LIN {X 0,Y 316.266,Z 772.149,A -85,B 0,C 180,E1 7195.232,E2 7195.232} C_VEL
LIN {X 0,Y 308.855,Z 793.821,A -85,B 0,C 180,E1 7194.701,E2 7194.701} C_VEL
LIN {X 0,Y 300.069,Z 815.244,A -85,B 0,C 180,E1 7194.002,E2 7194.002} C_VEL
LIN {X 0,Y 290.008,Z 835.58,A -85,B 0,C 180,E1 7193.134,E2 7193.134} C_VEL
LIN {X 0,Y 278.14,Z 856.299,A -85,B 0,C 180,E1 7191.998,E2 7191.998} C_VEL
LIN {X 0,Y 266.399,Z 874.047,A -85,B 0,C 180,E1 7190.75,E2 7190.75} C_VEL
LIN {X 0,Y 252.026,Z 893.205,A -85,B 0,C 180,E1 7189.023,E2 7189.023} C_VEL
LIN {X 0,Y 238.567,Z 909.092,A -85,B 0,C 180,E1 7187.167,E2 7187.167} C_VEL
LIN {X 0,Y 222.897,Z 925.612,A -85,B 0,C 180,E1 7184.652,E2 7184.652} C_VEL
LIN {X 0,Y 207.871,Z 939.883,A -85,B 0,C 180,E1 7181.782,E2 7181.782} C_VEL
LIN {X 0,Y 191.846,Z 953.573,A -85,B 0,C 180,E1 7178.064,E2 7178.064} C_VEL
LIN {X 0,Y 176.404,Z 965.739,A -85,B 0,C 180,E1 7173.567,E2 7173.567} C_VEL
LIN {X 0,Y 161.53,Z 976.411,A -85,B 0,C 180,E1 7167.988,E2 7167.988} C_VEL
LIN {X 0,Y 147.743,Z 985.877,A -85,B 0,C 180,E1 7160.997,E2 7160.997} C_VEL
LIN {X 0,Y 136.959,Z 993.036,A -85,B 0,C 180,E1 7153.329,E2 7153.329} C_VEL
LIN {X 0,Y 127.495,Z 999.606,A -85,B 0,C 180,E1 7142.954,E2 7142.954} C_VEL
LIN {X 0,Y 122.646,Z 1003.525,A -85,B 0,C 180,E1 7133.543,E2 7133.543} C_VEL
LIN {X 0,Y 120.303,Z 1006.266,A -85,B 0,C 180,E1 7122.968,E2 7122.968} C_VEL
LIN {X 0,Y 120.046,Z 1007.285,A -85,B 0,C 180,E1 7114.778,E2 7114.778} C_VEL
LIN {X 0,Y 120.078,Z 1007.432,A -85,B 0,C 180,E1 7108.093,E2 7108.093} C_VEL
LIN {X 0,Y 120.087,Z 1006.85,A -85,B 0,C 180,E1 7100.9,E2 7100.9} C_VEL
LIN {X 0,Y 121.024,Z 1005.17,A -85,B 0,C 180,E1 7092.204,E2 7092.204} C_VEL
LIN {X 0,Y 124.46,Z 1001.976,A -85,B 0,C 180,E1 7082.233,E2 7082.233} C_VEL
LIN {X 0,Y 131.486,Z 996.711,A -85,B 0,C 180,E1 7071.986,E2 7071.986} C_VEL
LIN {X 0,Y 141.32,Z 990.14,A -85,B 0,C 180,E1 7063.228,E2 7063.228} C_VEL
LIN {X 0,Y 153.783,Z 981.683,A -85,B 0,C 180,E1 7055.648,E2 7055.648} C_VEL
LIN {X 0,Y 168.407,Z 971.472,A -85,B 0,C 180,E1 7049.233,E2 7049.233} C_VEL
LIN {X 0,Y 183.206,Z 960.371,A -85,B 0,C 180,E1 7044.315,E2 7044.315} C_VEL
LIN {X 0,Y 199.948,Z 946.664,A -85,B 0,C 180,E1 7039.95,E2 7039.95} C_VEL
LIN {X 0,Y 215.947,Z 932.296,A -85,B 0,C 180,E1 7036.603,E2 7036.603} C_VEL
LIN {X 0,Y 231.694,Z 916.357,A -85,B 0,C 180,E1 7033.869,E2 7033.869} C_VEL
LIN {X 0,Y 247.003,Z 899.128,A -85,B 0,C 180,E1 7031.627,E2 7031.627} C_VEL
LIN {X 0,Y 260.107,Z 882.465,A -85,B 0,C 180,E1 7029.961,E2 7029.961} C_VEL
LIN {X 0,Y 274.246,Z 862.079,A -85,B 0,C 180,E1 7028.385,E2 7028.385} C_VEL
LIN {X 0,Y 285.918,Z 842.77,A -85,B 0,C 180,E1 7027.232,E2 7027.232} C_VEL
LIN {X 0,Y 296.695,Z 821.891,A -85,B 0,C 180,E1 7026.268,E2 7026.268} C_VEL
LIN {X 0,Y 305.842,Z 801.227,A -85,B 0,C 180,E1 7025.53,E2 7025.53} C_VEL
LIN {X 0,Y 313.42,Z 780.232,A -85,B 0,C 180,E1 7024.959,E2 7024.959} C_VEL
LIN {X 0,Y 320.064,Z 757.678,A -85,B 0,C 180,E1 7024.489,E2 7024.489} C_VEL
LIN {X 0,Y 325.022,Z 734.492,A -85,B 0,C 180,E1 7024.087,E2 7024.087} C_VEL
LIN {X 0,Y 329.208,Z 704.81,A -85,B 0,C 180,E1 7023.615,E2 7023.615} C_VEL
LIN {X 0,Y 337.766,Z 632.056,A -85,B 0,C 180,E1 7022.46,E2 7022.46} C_VEL
LIN {X 0,Y 337.614,Z 630.677,A -85,B 0,C 180,E1 7020.848,E2 7020.848} C_VEL
LIN {X 0,Y 337.652,Z 630.876,A -85,B 0,C 180,E1 7018.133,E2 7018.133} C_VEL
LIN {X 0,Y 337.738,Z 632.138,A -85,B 0,C 180,E1 7017.032,E2 7017.032} C_VEL
LIN {X 0,Y 326.503,Z 725.105,A -85,B 0,C 180,E1 7015.606,E2 7015.606} C_VEL
LIN {X 0,Y 321.976,Z 748.294,A -85,B 0,C 180,E1 7015.195,E2 7015.195} C_VEL
LIN {X 0,Y 316.268,Z 770.102,A -85,B 0,C 180,E1 7014.7,E2 7014.7} C_VEL
LIN {X 0,Y 308.91,Z 791.656,A -85,B 0,C 180,E1 7014.055,E2 7014.055} C_VEL
LIN {X 0,Y 300.013,Z 813.269,A -85,B 0,C 180,E1 7013.228,E2 7013.228} C_VEL
LIN {X 0,Y 290.069,Z 833.283,A -85,B 0,C 180,E1 7012.256,E2 7012.256} C_VEL
LIN {X 0,Y 277.932,Z 854.231,A -85,B 0,C 180,E1 7010.972,E2 7010.972} C_VEL
LIN {X 0,Y 266.23,Z 871.734,A -85,B 0,C 180,E1 7009.614,E2 7009.614} C_VEL
LIN {X 0,Y 252.131,Z 890.224,A -85,B 0,C 180,E1 7007.797,E2 7007.797} C_VEL
LIN {X 0,Y 238.696,Z 905.854,A -85,B 0,C 180,E1 7005.835,E2 7005.835} C_VEL
LIN {X 0,Y 223.399,Z 921.632,A -85,B 0,C 180,E1 7003.269,E2 7003.269} C_VEL
LIN {X 0,Y 208.189,Z 935.78,A -85,B 0,C 180,E1 7000.254,E2 7000.254} C_VEL
LIN {X 0,Y 192.815,Z 948.501,A -85,B 0,C 180,E1 6996.596,E2 6996.596} C_VEL
LIN {X 0,Y 177.595,Z 960.094,A -85,B 0,C 180,E1 6992.103,E2 6992.103} C_VEL
LIN {X 0,Y 162.895,Z 970.189,A -85,B 0,C 180,E1 6986.58,E2 6986.58} C_VEL
LIN {X 0,Y 148.728,Z 979.327,A -85,B 0,C 180,E1 6979.425,E2 6979.425} C_VEL
LIN {X 0,Y 137.676,Z 986.155,A -85,B 0,C 180,E1 6971.579,E2 6971.579} C_VEL
LIN {X 0,Y 128.644,Z 991.733,A -85,B 0,C 180,E1 6961.9,E2 6961.9} C_VEL
LIN {X 0,Y 123.386,Z 995.311,A -85,B 0,C 180,E1 6952.383,E2 6952.383} C_VEL
LIN {X 0,Y 120.711,Z 997.561,A -85,B 0,C 180,E1 6941.948,E2 6941.948} C_VEL
LIN {X 0,Y 120.131,Z 998.324,A -85,B 0,C 180,E1 6934.294,E2 6934.294} C_VEL
LIN {X 0,Y 120.104,Z 998.407,A -85,B 0,C 180,E1 6927.447,E2 6927.447} C_VEL
LIN {X 0,Y 120.477,Z 997.835,A -85,B 0,C 180,E1 6919.963,E2 6919.963} C_VEL
LIN {X 0,Y 122.224,Z 996.205,A -85,B 0,C 180,E1 6910.901,E2 6910.901} C_VEL
LIN {X 0,Y 127.095,Z 992.787,A -85,B 0,C 180,E1 6900.291,E2 6900.291} C_VEL
LIN {X 0,Y 134.407,Z 988.188,A -85,B 0,C 180,E1 6891.331,E2 6891.331} C_VEL
LIN {X 0,Y 146.095,Z 981.021,A -85,B 0,C 180,E1 6882.122,E2 6882.122} C_VEL
LIN {X 0,Y 158.918,Z 972.963,A -85,B 0,C 180,E1 6875.131,E2 6875.131} C_VEL
LIN {X 0,Y 173.157,Z 963.266,A -85,B 0,C 180,E1 6869.327,E2 6869.327} C_VEL
LIN {X 0,Y 188.062,Z 952.426,A -85,B 0,C 180,E1 6864.625,E2 6864.625} C_VEL
LIN {X 0,Y 203.368,Z 939.998,A -85,B 0,C 180,E1 6860.732,E2 6860.732} C_VEL
LIN {X 0,Y 219.042,Z 926.046,A -85,B 0,C 180,E1 6857.461,E2 6857.461} C_VEL
LIN {X 0,Y 233.766,Z 911.319,A -85,B 0,C 180,E1 6854.863,E2 6854.863} C_VEL
LIN {X 0,Y 249.373,Z 893.817,A -85,B 0,C 180,E1 6852.505,E2 6852.505} C_VEL
LIN {X 0,Y 262.598,Z 877.05,A -85,B 0,C 180,E1 6850.753,E2 6850.753} C_VEL
LIN {X 0,Y 275.882,Z 857.772,A -85,B 0,C 180,E1 6849.176,E2 6849.176} C_VEL
LIN {X 0,Y 287.669,Z 838.235,A -85,B 0,C 180,E1 6847.913,E2 6847.913} C_VEL
LIN {X 0,Y 298.071,Z 817.805,A -85,B 0,C 180,E1 6846.877,E2 6846.877} C_VEL
LIN {X 0,Y 307.128,Z 797.022,A -85,B 0,C 180,E1 6846.038,E2 6846.038} C_VEL
LIN {X 0,Y 314.556,Z 776.099,A -85,B 0,C 180,E1 6845.376,E2 6845.376} C_VEL
LIN {X 0,Y 321.052,Z 753.254,A -85,B 0,C 180,E1 6844.812,E2 6844.812} C_VEL
LIN {X 0,Y 325.588,Z 731.732,A -85,B 0,C 180,E1 6844.409,E2 6844.409} C_VEL
LIN {X 0,Y 329.863,Z 700.826,A -85,B 0,C 180,E1 6843.923,E2 6843.923} C_VEL
LIN {X 0,Y 337.962,Z 632.15,A -85,B 0,C 180,E1 6842.841,E2 6842.841} C_VEL
LIN {X 0,Y 337.832,Z 630.753,A -85,B 0,C 180,E1 6841.187,E2 6841.187} C_VEL
LIN {X 0,Y 337.856,Z 631.034,A -85,B 0,C 180,E1 6838.813,E2 6838.813} C_VEL
LIN {X 0,Y 337.961,Z 632.49,A -85,B 0,C 180,E1 6837.495,E2 6837.495} C_VEL
LIN {X 0,Y 326.742,Z 725.65,A -85,B 0,C 180,E1 6836.061,E2 6836.061} C_VEL
LIN {X 0,Y 325.489,Z 733.313,A -85,B 0,C 180,E1 6836.112,E2 6836.112} C_VEL
LIN {X 0,Y 321.09,Z 752.516,A -85,B 0,C 180,E1 6836.86,E2 6836.86} C_VEL
LIN {X 0,Y 319.042,Z 760.005,A -85,B 0,C 180,E1 6836.907,E2 6836.907} C_VEL
LIN {X 0,Y 312.512,Z 781.566,A -85,B 0,C 180,E1 6836.481,E2 6836.481} C_VEL
LIN {X 0,Y 304.202,Z 803.689,A -85,B 0,C 180,E1 6835.902,E2 6835.902} C_VEL
LIN {X 0,Y 295.301,Z 823.326,A -85,B 0,C 180,E1 6835.234,E2 6835.234} C_VEL
LIN {X 0,Y 283.842,Z 844.807,A -85,B 0,C 180,E1 6834.282,E2 6834.282} C_VEL
LIN {X 0,Y 272.338,Z 863.402,A -85,B 0,C 180,E1 6833.22,E2 6833.22} C_VEL
LIN {X 0,Y 258.312,Z 883.078,A -85,B 0,C 180,E1 6831.766,E2 6831.766} C_VEL
LIN {X 0,Y 244.323,Z 900.449,A -85,B 0,C 180,E1 6830.103,E2 6830.103} C_VEL
LIN {X 0,Y 228.952,Z 917.166,A -85,B 0,C 180,E1 6827.995,E2 6827.995} C_VEL
LIN {X 0,Y 212.846,Z 932.917,A -85,B 0,C 180,E1 6825.376,E2 6825.376} C_VEL
LIN {X 0,Y 197.001,Z 946.701,A -85,B 0,C 180,E1 6822.271,E2 6822.271} C_VEL
LIN {X 0,Y 179.129,Z 960.742,A -85,B 0,C 180,E1 6817.893,E2 6817.893} C_VEL
LIN {X 0,Y 163.006,Z 972.297,A -85,B 0,C 180,E1 6812.788,E2 6812.788} C_VEL
LIN {X 0,Y 148.399,Z 981.854,A -85,B 0,C 180,E1 6806.656,E2 6806.656} C_VEL
LIN {X 0,Y 135.173,Z 990.205,A -85,B 0,C 180,E1 6798.974,E2 6798.974} C_VEL
LIN {X 0,Y 124.603,Z 996.704,A -85,B 0,C 180,E1 6789.933,E2 6789.933} C_VEL
LIN {X 0,Y 116.938,Z 1001.86,A -85,B 0,C 180,E1 6779.166,E2 6779.166} C_VEL
LIN {X 0,Y 113.251,Z 1004.881,A -85,B 0,C 180,E1 6769.065,E2 6769.065} C_VEL
LIN {X 0,Y 112.105,Z 1006.557,A -85,B 0,C 180,E1 6759.757,E2 6759.757} C_VEL
LIN {X 0,Y 112.078,Z 1007.135,A -85,B 0,C 180,E1 6752.046,E2 6752.046} C_VEL
LIN {X 0,Y 112.05,Z 1007.006,A -85,B 0,C 180,E1 6745.396,E2 6745.396} C_VEL
LIN {X 0,Y 112.287,Z 1006.1,A -85,B 0,C 180,E1 6737.14,E2 6737.14} C_VEL
LIN {X 0,Y 114.575,Z 1003.697,A -85,B 0,C 180,E1 6726.337,E2 6726.337} C_VEL
LIN {X 0,Y 119.811,Z 999.777,A -85,B 0,C 180,E1 6716.01,E2 6716.01} C_VEL
LIN {X 0,Y 129.046,Z 993.932,A -85,B 0,C 180,E1 6705.795,E2 6705.795} C_VEL
LIN {X 0,Y 140.886,Z 986.539,A -85,B 0,C 180,E1 6697.369,E2 6697.369} C_VEL
LIN {X 0,Y 155.828,Z 976.963,A -85,B 0,C 180,E1 6689.992,E2 6689.992} C_VEL
LIN {X 0,Y 170.862,Z 966.695,A -85,B 0,C 180,E1 6684.549,E2 6684.549} C_VEL
LIN {X 0,Y 187.219,Z 954.442,A -85,B 0,C 180,E1 6679.979,E2 6679.979} C_VEL
LIN {X 0,Y 203.246,Z 941.356,A -85,B 0,C 180,E1 6676.43,E2 6676.43} C_VEL
LIN {X 0,Y 219.044,Z 926.852,A -85,B 0,C 180,E1 6673.555,E2 6673.555} C_VEL
LIN {X 0,Y 234.828,Z 910.851,A -85,B 0,C 180,E1 6671.157,E2 6671.157} C_VEL
LIN {X 0,Y 249.198,Z 894.325,A -85,B 0,C 180,E1 6669.284,E2 6669.284} C_VEL
LIN {X 0,Y 263.299,Z 876.152,A -85,B 0,C 180,E1 6667.692,E2 6667.692} C_VEL
LIN {X 0,Y 275.195,Z 858.637,A -85,B 0,C 180,E1 6666.497,E2 6666.497} C_VEL
LIN {X 0,Y 287.593,Z 837.788,A -85,B 0,C 180,E1 6665.386,E2 6665.386} C_VEL
LIN {X 0,Y 297.375,Z 818.548,A -85,B 0,C 180,E1 6664.591,E2 6664.591} C_VEL
LIN {X 0,Y 307.119,Z 795.819,A -85,B 0,C 180,E1 6663.871,E2 6663.871} C_VEL
LIN {X 0,Y 314.464,Z 774.962,A -85,B 0,C 180,E1 6663.381,E2 6663.381} C_VEL
LIN {X 0,Y 320.903,Z 751.526,A -85,B 0,C 180,E1 6662.952,E2 6662.952} C_VEL
LIN {X 0,Y 325.664,Z 728.122,A -85,B 0,C 180,E1 6662.575,E2 6662.575} C_VEL
LIN {X 0,Y 333.582,Z 664.479,A -85,B 0,C 180,E1 6661.619,E2 6661.619} C_VEL
LIN {X 0,Y 336.658,Z 638.896,A -85,B 0,C 180,E1 6661.238,E2 6661.238} C_VEL
LIN {X 0,Y 336.651,Z 638.631,A -85,B 0,C 180,E1 6658.468,E2 6658.468} C_VEL
LIN {X 0,Y 336.625,Z 639.037,A -85,B 0,C 180,E1 6658.292,E2 6658.292} C_VEL
LIN {X 0,Y 325.971,Z 725.542,A -85,B 0,C 180,E1 6657.007,E2 6657.007} C_VEL
LIN {X 0,Y 321.363,Z 748.782,A -85,B 0,C 180,E1 6656.614,E2 6656.614} C_VEL
LIN {X 0,Y 315.386,Z 771.203,A -85,B 0,C 180,E1 6656.129,E2 6656.129} C_VEL
LIN {X 0,Y 307.862,Z 792.809,A -85,B 0,C 180,E1 6655.513,E2 6655.513} C_VEL
LIN {X 0,Y 298.689,Z 814.575,A -85,B 0,C 180,E1 6654.718,E2 6654.718} C_VEL
LIN {X 0,Y 289.148,Z 833.487,A -85,B 0,C 180,E1 6653.846,E2 6653.846} C_VEL
LIN {X 0,Y 277.193,Z 853.902,A -85,B 0,C 180,E1 6652.668,E2 6652.668} C_VEL
LIN {X 0,Y 265.593,Z 871.045,A -85,B 0,C 180,E1 6651.423,E2 6651.423} C_VEL
LIN {X 0,Y 250.944,Z 890.046,A -85,B 0,C 180,E1 6649.671,E2 6649.671} C_VEL
LIN {X 0,Y 237.279,Z 905.664,A -85,B 0,C 180,E1 6647.82,E2 6647.82} C_VEL
LIN {X 0,Y 221.178,Z 921.943,A -85,B 0,C 180,E1 6645.304,E2 6645.304} C_VEL
LIN {X 0,Y 205.555,Z 936.091,A -85,B 0,C 180,E1 6642.412,E2 6642.412} C_VEL
LIN {X 0,Y 189.689,Z 948.813,A -85,B 0,C 180,E1 6638.884,E2 6638.884} C_VEL
LIN {X 0,Y 173.466,Z 960.676,A -85,B 0,C 180,E1 6634.386,E2 6634.386} C_VEL
LIN {X 0,Y 158.488,Z 970.501,A -85,B 0,C 180,E1 6629.078,E2 6629.078} C_VEL
LIN {X 0,Y 143.483,Z 979.639,A -85,B 0,C 180,E1 6621.936,E2 6621.936} C_VEL
LIN {X 0,Y 131.907,Z 986.289,A -85,B 0,C 180,E1 6614.208,E2 6614.208} C_VEL
LIN {X 0,Y 121.743,Z 992.042,A -85,B 0,C 180,E1 6603.944,E2 6603.944} C_VEL
LIN {X 0,Y 115.678,Z 995.769,A -85,B 0,C 180,E1 6593.424,E2 6593.424} C_VEL
LIN {X 0,Y 112.747,Z 997.926,A -85,B 0,C 180,E1 6582.286,E2 6582.286} C_VEL
LIN {X 0,Y 112.13,Z 998.645,A -85,B 0,C 180,E1 6574.089,E2 6574.089} C_VEL
LIN {X 0,Y 112.111,Z 998.693,A -85,B 0,C 180,E1 6566.932,E2 6566.932} C_VEL
LIN {X 0,Y 112.615,Z 998.074,A -85,B 0,C 180,E1 6558.736,E2 6558.736} C_VEL
LIN {X 0,Y 114.863,Z 996.318,A -85,B 0,C 180,E1 6548.659,E2 6548.659} C_VEL
LIN {X 0,Y 120.677,Z 992.7,A -85,B 0,C 180,E1 6537.418,E2 6537.418} C_VEL
LIN {X 0,Y 129.445,Z 987.765,A -85,B 0,C 180,E1 6527.782,E2 6527.782} C_VEL
LIN {X 0,Y 141.035,Z 981.12,A -85,B 0,C 180,E1 6519.405,E2 6519.405} C_VEL
LIN {X 0,Y 154.975,Z 972.87,A -85,B 0,C 180,E1 6512.317,E2 6512.317} C_VEL
LIN {X 0,Y 170.554,Z 962.706,A -85,B 0,C 180,E1 6506.459,E2 6506.459} C_VEL
LIN {X 0,Y 187.448,Z 950.662,A -85,B 0,C 180,E1 6501.596,E2 6501.596} C_VEL
LIN {X 0,Y 202.93,Z 938.41,A -85,B 0,C 180,E1 6498.04,E2 6498.04} C_VEL
LIN {X 0,Y 219.351,Z 923.853,A -85,B 0,C 180,E1 6494.928,E2 6494.928} C_VEL
LIN {X 0,Y 234.51,Z 908.883,A -85,B 0,C 180,E1 6492.508,E2 6492.508} C_VEL
LIN {X 0,Y 249.101,Z 892.492,A -85,B 0,C 180,E1 6490.487,E2 6490.487} C_VEL
LIN {X 0,Y 263.029,Z 874.979,A -85,B 0,C 180,E1 6488.795,E2 6488.795} C_VEL
LIN {X 0,Y 275.495,Z 856.858,A -85,B 0,C 180,E1 6487.427,E2 6487.427} C_VEL
LIN {X 0,Y 287.623,Z 836.758,A -85,B 0,C 180,E1 6486.222,E2 6486.222} C_VEL
LIN {X 0,Y 297.695,Z 817.103,A -85,B 0,C 180,E1 6485.292,E2 6485.292} C_VEL
LIN {X 0,Y 307.352,Z 794.763,A -85,B 0,C 180,E1 6484.456,E2 6484.456} C_VEL
LIN {X 0,Y 314.635,Z 774.182,A -85,B 0,C 180,E1 6483.858,E2 6483.858} C_VEL
LIN {X 0,Y 321.12,Z 750.814,A -85,B 0,C 180,E1 6483.333,E2 6483.333} C_VEL
LIN {X 0,Y 325.756,Z 728.384,A -85,B 0,C 180,E1 6482.945,E2 6482.945} C_VEL
LIN {X 0,Y 331.088,Z 687.088,A -85,B 0,C 180,E1 6482.326,E2 6482.326} C_VEL
LIN {X 0,Y 336.866,Z 639.033,A -85,B 0,C 180,E1 6481.616,E2 6481.616} C_VEL
LIN {X 0,Y 336.813,Z 638.685,A -85,B 0,C 180,E1 6480.341,E2 6480.341} C_VEL
LIN {X 0,Y 336.865,Z 638.921,A -85,B 0,C 180,E1 6478.98,E2 6478.98} C_VEL
LIN {X 0,Y 336.84,Z 639.386,A -85,B 0,C 180,E1 6478.753,E2 6478.753} C_VEL
LIN {X 0,Y 326.086,Z 726.797,A -85,B 0,C 180,E1 6477.449,E2 6477.449} C_VEL
LIN {X 0,Y 321.403,Z 750.38,A -85,B 0,C 180,E1 6477.07,E2 6477.07} C_VEL
LIN {X 0,Y 319.042,Z 760.005,A -85,B 0,C 180,E1 6476.907,E2 6476.907} C_VEL
LIN {X 0,Y 316.878,Z 767.449,A -85,B 0,C 180,E1 6476.972,E2 6476.972} C_VEL
LIN {X 0,Y 310.535,Z 786.139,A -85,B 0,C 180,E1 6477.715,E2 6477.715} C_VEL
LIN {X 0,Y 307.729,Z 793.374,A -85,B 0,C 180,E1 6477.693,E2 6477.693} C_VEL
LIN {X 0,Y 298.319,Z 815.659,A -85,B 0,C 180,E1 6477.06,E2 6477.06} C_VEL
LIN {X 0,Y 287.888,Z 836.146,A -85,B 0,C 180,E1 6476.293,E2 6476.293} C_VEL
LIN {X 0,Y 275.37,Z 857.177,A -85,B 0,C 180,E1 6475.271,E2 6475.271} C_VEL
LIN {X 0,Y 263.298,Z 874.788,A -85,B 0,C 180,E1 6474.168,E2 6474.168} C_VEL
LIN {X 0,Y 248.44,Z 893.744,A -85,B 0,C 180,E1 6472.633,E2 6472.633} C_VEL
LIN {X 0,Y 233.89,Z 910.186,A -85,B 0,C 180,E1 6470.896,E2 6470.896} C_VEL
LIN {X 0,Y 218.171,Z 925.852,A -85,B 0,C 180,E1 6468.707,E2 6468.707} C_VEL
LIN {X 0,Y 201.946,Z 940.437,A -85,B 0,C 180,E1 6466.006,E2 6466.006} C_VEL
LIN {X 0,Y 185.391,Z 953.598,A -85,B 0,C 180,E1 6462.651,E2 6462.651} C_VEL
LIN {X 0,Y 168.796,Z 965.657,A -85,B 0,C 180,E1 6458.418,E2 6458.418} C_VEL
LIN {X 0,Y 152.555,Z 976.256,A -85,B 0,C 180,E1 6453.033,E2 6453.033} C_VEL
LIN {X 0,Y 136.223,Z 986.138,A -85,B 0,C 180,E1 6445.587,E2 6445.587} C_VEL
LIN {X 0,Y 123.707,Z 993.354,A -85,B 0,C 180,E1 6437.344,E2 6437.344} C_VEL
LIN {X 0,Y 113.385,Z 999.281,A -85,B 0,C 180,E1 6426.841,E2 6426.841} C_VEL
LIN {X 0,Y 107.072,Z 1003.414,A -85,B 0,C 180,E1 6415.438,E2 6415.438} C_VEL
LIN {X 0,Y 104.375,Z 1005.806,A -85,B 0,C 180,E1 6403.856,E2 6403.856} C_VEL
LIN {X 0,Y 104.052,Z 1006.683,A -85,B 0,C 180,E1 6395.515,E2 6395.515} C_VEL
LIN {X 0,Y 104.089,Z 1006.856,A -85,B 0,C 180,E1 6388.35,E2 6388.35} C_VEL
LIN {X 0,Y 104.111,Z 1006.317,A -85,B 0,C 180,E1 6380.048,E2 6380.048} C_VEL
LIN {X 0,Y 105.449,Z 1004.632,A -85,B 0,C 180,E1 6369.832,E2 6369.832} C_VEL
LIN {X 0,Y 109.774,Z 1001.524,A -85,B 0,C 180,E1 6358.729,E2 6358.729} C_VEL
LIN {X 0,Y 118.314,Z 996.349,A -85,B 0,C 180,E1 6347.471,E2 6347.471} C_VEL
LIN {X 0,Y 129.819,Z 989.838,A -85,B 0,C 180,E1 6338.234,E2 6338.234} C_VEL
LIN {X 0,Y 144.314,Z 981.246,A -85,B 0,C 180,E1 6330.381,E2 6330.381} C_VEL
LIN {X 0,Y 160.106,Z 971.367,A -85,B 0,C 180,E1 6324.267,E2 6324.267} C_VEL
LIN {X 0,Y 176.214,Z 960.271,A -85,B 0,C 180,E1 6319.558,E2 6319.558} C_VEL
LIN {X 0,Y 194.006,Z 946.747,A -85,B 0,C 180,E1 6315.501,E2 6315.501} C_VEL
LIN {X 0,Y 209.984,Z 933.235,A -85,B 0,C 180,E1 6312.578,E2 6312.578} C_VEL
LIN {X 0,Y 226.436,Z 917.606,A -85,B 0,C 180,E1 6310.082,E2 6310.082} C_VEL
LIN {X 0,Y 242.221,Z 900.853,A -85,B 0,C 180,E1 6308.067,E2 6308.067} C_VEL
LIN {X 0,Y 256.572,Z 883.384,A -85,B 0,C 180,E1 6306.483,E2 6306.483} C_VEL
LIN {X 0,Y 270.517,Z 864.252,A -85,B 0,C 180,E1 6305.144,E2 6305.144} C_VEL
LIN {X 0,Y 282.65,Z 844.958,A -85,B 0,C 180,E1 6304.106,E2 6304.106} C_VEL
LIN {X 0,Y 294.383,Z 823.291,A -85,B 0,C 180,E1 6303.208,E2 6303.208} C_VEL
LIN {X 0,Y 303.531,Z 803.322,A -85,B 0,C 180,E1 6302.578,E2 6302.578} C_VEL
LIN {X 0,Y 312.113,Z 780.59,A -85,B 0,C 180,E1 6302.031,E2 6302.031} C_VEL
LIN {X 0,Y 318.826,Z 758.475,A -85,B 0,C 180,E1 6301.63,E2 6301.63} C_VEL
LIN {X 0,Y 324.028,Z 735.143,A -85,B 0,C 180,E1 6301.268,E2 6301.268} C_VEL
LIN {X 0,Y 327.89,Z 709.899,A -85,B 0,C 180,E1 6300.895,E2 6300.895} C_VEL
LIN {X 0,Y 335.601,Z 646.557,A -85,B 0,C 180,E1 6299.957,E2 6299.957} C_VEL
LIN {X 0,Y 335.578,Z 646.733,A -85,B 0,C 180,E1 6299.549,E2 6299.549} C_VEL
LIN {X 0,Y 325.615,Z 726.115,A -85,B 0,C 180,E1 6298.408,E2 6298.408} C_VEL
LIN {X 0,Y 320.96,Z 749.221,A -85,B 0,C 180,E1 6298.038,E2 6298.038} C_VEL
LIN {X 0,Y 314.946,Z 771.513,A -85,B 0,C 180,E1 6297.585,E2 6297.585} C_VEL
LIN {X 0,Y 307.338,Z 793.118,A -85,B 0,C 180,E1 6297.005,E2 6297.005} C_VEL
LIN {X 0,Y 298.056,Z 814.883,A -85,B 0,C 180,E1 6296.259,E2 6296.259} C_VEL
LIN {X 0,Y 288.207,Z 834.142,A -85,B 0,C 180,E1 6295.423,E2 6295.423} C_VEL
LIN {X 0,Y 275.796,Z 854.938,A -85,B 0,C 180,E1 6294.288,E2 6294.288} C_VEL
LIN {X 0,Y 263.845,Z 872.27,A -85,B 0,C 180,E1 6293.093,E2 6293.093} C_VEL
LIN {X 0,Y 249.193,Z 890.845,A -85,B 0,C 180,E1 6291.462,E2 6291.462} C_VEL
LIN {X 0,Y 235.395,Z 906.294,A -85,B 0,C 180,E1 6289.723,E2 6289.723} C_VEL
LIN {X 0,Y 219.24,Z 922.253,A -85,B 0,C 180,E1 6287.379,E2 6287.379} C_VEL
LIN {X 0,Y 202.94,Z 936.645,A -85,B 0,C 180,E1 6284.57,E2 6284.57} C_VEL
LIN {X 0,Y 186.035,Z 949.747,A -85,B 0,C 180,E1 6281.05,E2 6281.05} C_VEL
LIN {X 0,Y 168.895,Z 961.723,A -85,B 0,C 180,E1 6276.56,E2 6276.56} C_VEL
LIN {X 0,Y 153.669,Z 971.26,A -85,B 0,C 180,E1 6271.434,E2 6271.434} C_VEL
LIN {X 0,Y 137.893,Z 980.292,A -85,B 0,C 180,E1 6264.291,E2 6264.291} C_VEL
LIN {X 0,Y 125.059,Z 987.184,A -85,B 0,C 180,E1 6256.009,E2 6256.009} C_VEL
LIN {X 0,Y 114.63,Z 992.548,A -85,B 0,C 180,E1 6245.755,E2 6245.755} C_VEL
LIN {X 0,Y 108.011,Z 996.227,A -85,B 0,C 180,E1 6234.613,E2 6234.613} C_VEL
LIN {X 0,Y 104.861,Z 998.23,A -85,B 0,C 180,E1 6223.226,E2 6223.226} C_VEL
LIN {X 0,Y 104.144,Z 998.945,A -85,B 0,C 180,E1 6214.403,E2 6214.403} C_VEL
LIN {X 0,Y 104.115,Z 999.011,A -85,B 0,C 180,E1 6207.157,E2 6207.157} C_VEL
LIN {X 0,Y 104.644,Z 998.439,A -85,B 0,C 180,E1 6198.425,E2 6198.425} C_VEL
LIN {X 0,Y 106.963,Z 996.815,A -85,B 0,C 180,E1 6188.044,E2 6188.044} C_VEL
LIN {X 0,Y 113.478,Z 993.205,A -85,B 0,C 180,E1 6175.676,E2 6175.676} C_VEL
LIN {X 0,Y 122.762,Z 988.409,A -85,B 0,C 180,E1 6165.787,E2 6165.787} C_VEL
LIN {X 0,Y 135.93,Z 981.429,A -85,B 0,C 180,E1 6156.708,E2 6156.708} C_VEL
LIN {X 0,Y 150.708,Z 973.18,A -85,B 0,C 180,E1 6149.655,E2 6149.655} C_VEL
LIN {X 0,Y 166.463,Z 963.38,A -85,B 0,C 180,E1 6144.091,E2 6144.091} C_VEL
LIN {X 0,Y 183.458,Z 951.798,A -85,B 0,C 180,E1 6139.478,E2 6139.478} C_VEL
LIN {X 0,Y 199.661,Z 939.405,A -85,B 0,C 180,E1 6135.971,E2 6135.971} C_VEL
LIN {X 0,Y 216.482,Z 924.991,A -85,B 0,C 180,E1 6132.982,E2 6132.982} C_VEL
LIN {X 0,Y 231.032,Z 911.013,A -85,B 0,C 180,E1 6130.794,E2 6130.794} C_VEL
LIN {X 0,Y 246.809,Z 893.891,A -85,B 0,C 180,E1 6128.745,E2 6128.745} C_VEL
LIN {X 0,Y 260.495,Z 877.096,A -85,B 0,C 180,E1 6127.186,E2 6127.186} C_VEL
LIN {X 0,Y 273.844,Z 858.251,A -85,B 0,C 180,E1 6125.82,E2 6125.82} C_VEL
LIN {X 0,Y 285.893,Z 838.83,A -85,B 0,C 180,E1 6124.705,E2 6124.705} C_VEL
LIN {X 0,Y 296.573,Z 818.397,A -85,B 0,C 180,E1 6123.785,E2 6123.785} C_VEL
LIN {X 0,Y 305.855,Z 797.609,A -85,B 0,C 180,E1 6123.041,E2 6123.041} C_VEL
LIN {X 0,Y 313.46,Z 776.682,A -85,B 0,C 180,E1 6122.454,E2 6122.454} C_VEL
LIN {X 0,Y 320.107,Z 753.828,A -85,B 0,C 180,E1 6121.955,E2 6121.955} C_VEL
LIN {X 0,Y 324.744,Z 732.332,A -85,B 0,C 180,E1 6121.592,E2 6121.592} C_VEL
LIN {X 0,Y 329.15,Z 701.421,A -85,B 0,C 180,E1 6121.143,E2 6121.143} C_VEL
LIN {X 0,Y 335.838,Z 646.625,A -85,B 0,C 180,E1 6120.342,E2 6120.342} C_VEL
LIN {X 0,Y 335.823,Z 646.762,A -85,B 0,C 180,E1 6120.013,E2 6120.013} C_VEL
LIN {X 0,Y 325.796,Z 726.732,A -85,B 0,C 180,E1 6118.859,E2 6118.859} C_VEL
LIN {X 0,Y 321.061,Z 750.221,A -85,B 0,C 180,E1 6118.503,E2 6118.503} C_VEL
LIN {X 0,Y 314.841,Z 773.107,A -85,B 0,C 180,E1 6118.121,E2 6118.121} C_VEL
LIN {X 0,Y 307.729,Z 793.374,A -85,B 0,C 180,E1 6117.693,E2 6117.693} C_VEL
LIN {X 0,Y 304.825,Z 800.733,A -85,B 0,C 180,E1 6117.696,E2 6117.696} C_VEL
LIN {X 0,Y 296.433,Z 818.686,A -85,B 0,C 180,E1 6118.323,E2 6118.323} C_VEL
LIN {X 0,Y 293.03,Z 825.52,A -85,B 0,C 180,E1 6118.289,E2 6118.289} C_VEL
LIN {X 0,Y 281.699,Z 845.84,A -85,B 0,C 180,E1 6117.498,E2 6117.498} C_VEL
LIN {X 0,Y 269.426,Z 865.02,A -85,B 0,C 180,E1 6116.534,E2 6116.534} C_VEL
LIN {X 0,Y 255.784,Z 883.345,A -85,B 0,C 180,E1 6115.336,E2 6115.336} C_VEL
LIN {X 0,Y 241.318,Z 900.647,A -85,B 0,C 180,E1 6113.876,E2 6113.876} C_VEL
LIN {X 0,Y 226.089,Z 916.551,A -85,B 0,C 180,E1 6112.104,E2 6112.104} C_VEL
LIN {X 0,Y 209.266,Z 932.298,A -85,B 0,C 180,E1 6109.787,E2 6109.787} C_VEL
LIN {X 0,Y 192.851,Z 945.859,A -85,B 0,C 180,E1 6107.061,E2 6107.061} C_VEL
LIN {X 0,Y 174.376,Z 959.531,A -85,B 0,C 180,E1 6103.23,E2 6103.23} C_VEL
LIN {X 0,Y 157.664,Z 970.617,A -85,B 0,C 180,E1 6098.771,E2 6098.771} C_VEL
LIN {X 0,Y 140.604,Z 980.809,A -85,B 0,C 180,E1 6092.724,E2 6092.724} C_VEL
LIN {X 0,Y 125.448,Z 989.255,A -85,B 0,C 180,E1 6085.172,E2 6085.172} C_VEL
LIN {X 0,Y 112.81,Z 995.813,A -85,B 0,C 180,E1 6075.878,E2 6075.878} C_VEL
LIN {X 0,Y 103.103,Z 1001.069,A -85,B 0,C 180,E1 6064.224,E2 6064.224} C_VEL
LIN {X 0,Y 97.896,Z 1004.267,A -85,B 0,C 180,E1 6052.203,E2 6052.203} C_VEL
LIN {X 0,Y 96.142,Z 1006.024,A -85,B 0,C 180,E1 6040.79,E2 6040.79} C_VEL
LIN {X 0,Y 96.09,Z 1006.559,A -85,B 0,C 180,E1 6031.79,E2 6031.79} C_VEL
LIN {X 0,Y 96.056,Z 1006.378,A -85,B 0,C 180,E1 6024.028,E2 6024.028} C_VEL
LIN {X 0,Y 96.655,Z 1005.339,A -85,B 0,C 180,E1 6013.785,E2 6013.785} C_VEL
LIN {X 0,Y 100.428,Z 1002.57,A -85,B 0,C 180,E1 6000.807,E2 6000.807} C_VEL
LIN {X 0,Y 107.673,Z 998.499,A -85,B 0,C 180,E1 5989.464,E2 5989.464} C_VEL
LIN {X 0,Y 119.923,Z 992.042,A -85,B 0,C 180,E1 5978.407,E2 5978.407} C_VEL
LIN {X 0,Y 134.134,Z 984.446,A -85,B 0,C 180,E1 5970.167,E2 5970.167} C_VEL
LIN {X 0,Y 150.481,Z 974.917,A -85,B 0,C 180,E1 5963.537,E2 5963.537} C_VEL
LIN {X 0,Y 167.63,Z 964.065,A -85,B 0,C 180,E1 5958.428,E2 5958.428} C_VEL
LIN {X 0,Y 184.827,Z 951.867,A -85,B 0,C 180,E1 5954.486,E2 5954.486} C_VEL
LIN {X 0,Y 202.817,Z 937.619,A -85,B 0,C 180,E1 5951.213,E2 5951.213} C_VEL
LIN {X 0,Y 218.557,Z 923.65,A -85,B 0,C 180,E1 5948.872,E2 5948.872} C_VEL
LIN {X 0,Y 235.568,Z 906.583,A -85,B 0,C 180,E1 5946.747,E2 5946.747} C_VEL
LIN {X 0,Y 250.936,Z 889.204,A -85,B 0,C 180,E1 5945.124,E2 5945.124} C_VEL
LIN {X 0,Y 265.019,Z 870.811,A -85,B 0,C 180,E1 5943.825,E2 5943.825} C_VEL
LIN {X 0,Y 278.248,Z 851.184,A -85,B 0,C 180,E1 5942.756,E2 5942.756} C_VEL
LIN {X 0,Y 289.093,Z 832.457,A -85,B 0,C 180,E1 5941.968,E2 5941.968} C_VEL
LIN {X 0,Y 299.495,Z 811.656,A -85,B 0,C 180,E1 5941.284,E2 5941.284} C_VEL
LIN {X 0,Y 307.946,Z 791.327,A -85,B 0,C 180,E1 5940.768,E2 5940.768} C_VEL
LIN {X 0,Y 316.077,Z 767.298,A -85,B 0,C 180,E1 5940.322,E2 5940.322} C_VEL
LIN {X 0,Y 321.822,Z 745.271,A -85,B 0,C 180,E1 5939.994,E2 5939.994} C_VEL
LIN {X 0,Y 324.885,Z 729.953,A -85,B 0,C 180,E1 5939.766,E2 5939.766} C_VEL
LIN {X 0,Y 320.244,Z 751.796,A -85,B 0,C 180,E1 5939.428,E2 5939.428} C_VEL
LIN {X 0,Y 313.717,Z 774.768,A -85,B 0,C 180,E1 5938.974,E2 5938.974} C_VEL
LIN {X 0,Y 306.528,Z 794.705,A -85,B 0,C 180,E1 5938.466,E2 5938.466} C_VEL
LIN {X 0,Y 296.501,Z 817.496,A -85,B 0,C 180,E1 5937.721,E2 5937.721} C_VEL
LIN {X 0,Y 286.338,Z 836.888,A -85,B 0,C 180,E1 5936.916,E2 5936.916} C_VEL
LIN {X 0,Y 274.135,Z 856.703,A -85,B 0,C 180,E1 5935.881,E2 5935.881} C_VEL
LIN {X 0,Y 261.547,Z 874.561,A -85,B 0,C 180,E1 5934.705,E2 5934.705} C_VEL
LIN {X 0,Y 247.163,Z 892.248,A -85,B 0,C 180,E1 5933.219,E2 5933.219} C_VEL
LIN {X 0,Y 232.092,Z 908.708,A -85,B 0,C 180,E1 5931.44,E2 5931.44} C_VEL
LIN {X 0,Y 215.753,Z 924.228,A -85,B 0,C 180,E1 5929.216,E2 5929.216} C_VEL
LIN {X 0,Y 198.503,Z 938.824,A -85,B 0,C 180,E1 5926.412,E2 5926.412} C_VEL
LIN {X 0,Y 182.657,Z 950.681,A -85,B 0,C 180,E1 5923.299,E2 5923.299} C_VEL
LIN {X 0,Y 164.141,Z 963.04,A -85,B 0,C 180,E1 5918.728,E2 5918.728} C_VEL
LIN {X 0,Y 147.961,Z 972.704,A -85,B 0,C 180,E1 5913.512,E2 5913.512} C_VEL
LIN {X 0,Y 132.556,Z 980.945,A -85,B 0,C 180,E1 5906.84,E2 5906.84} C_VEL
LIN {X 0,Y 118.689,Z 987.899,A -85,B 0,C 180,E1 5898.277,E2 5898.277} C_VEL
LIN {X 0,Y 107.646,Z 993.054,A -85,B 0,C 180,E1 5887.802,E2 5887.802} C_VEL
LIN {X 0,Y 100.153,Z 996.766,A -85,B 0,C 180,E1 5875.417,E2 5875.417} C_VEL
LIN {X 0,Y 96.915,Z 998.595,A -85,B 0,C 180,E1 5863.723,E2 5863.723} C_VEL
LIN {X 0,Y 96.141,Z 999.266,A -85,B 0,C 180,E1 5854.173,E2 5854.173} C_VEL
LIN {X 0,Y 96.127,Z 999.294,A -85,B 0,C 180,E1 5846.421,E2 5846.421} C_VEL
LIN {X 0,Y 96.821,Z 998.68,A -85,B 0,C 180,E1 5836.868,E2 5836.868} C_VEL
LIN {X 0,Y 99.662,Z 997.015,A -85,B 0,C 180,E1 5825.713,E2 5825.713} C_VEL
LIN {X 0,Y 107.19,Z 993.315,A -85,B 0,C 180,E1 5812.68,E2 5812.68} C_VEL
LIN {X 0,Y 117.734,Z 988.383,A -85,B 0,C 180,E1 5802.372,E2 5802.372} C_VEL
LIN {X 0,Y 131.15,Z 981.738,A -85,B 0,C 180,E1 5793.807,E2 5793.807} C_VEL
LIN {X 0,Y 146.788,Z 973.489,A -85,B 0,C 180,E1 5786.845,E2 5786.845} C_VEL
LIN {X 0,Y 163.26,Z 963.688,A -85,B 0,C 180,E1 5781.439,E2 5781.439} C_VEL
LIN {X 0,Y 180.873,Z 952.106,A -85,B 0,C 180,E1 5777.012,E2 5777.012} C_VEL
LIN {X 0,Y 197.554,Z 939.711,A -85,B 0,C 180,E1 5773.676,E2 5773.676} C_VEL
LIN {X 0,Y 214.787,Z 925.296,A -85,B 0,C 180,E1 5770.849,E2 5770.849} C_VEL
LIN {X 0,Y 229.906,Z 911.059,A -85,B 0,C 180,E1 5768.756,E2 5768.756} C_VEL
LIN {X 0,Y 245.702,Z 894.193,A -85,B 0,C 180,E1 5766.866,E2 5766.866} C_VEL
LIN {X 0,Y 259.592,Z 877.412,A -85,B 0,C 180,E1 5765.409,E2 5765.409} C_VEL
LIN {X 0,Y 272.656,Z 859.279,A -85,B 0,C 180,E1 5764.173,E2 5764.173} C_VEL
LIN {X 0,Y 284.854,Z 839.945,A -85,B 0,C 180,E1 5763.128,E2 5763.128} C_VEL
LIN {X 0,Y 295.731,Z 819.544,A -85,B 0,C 180,E1 5762.262,E2 5762.262} C_VEL
LIN {X 0,Y 305.311,Z 798.477,A -85,B 0,C 180,E1 5761.552,E2 5761.552} C_VEL
LIN {X 0,Y 313.219,Z 776.974,A -85,B 0,C 180,E1 5760.988,E2 5760.988} C_VEL
LIN {X 0,Y 319.934,Z 754.116,A -85,B 0,C 180,E1 5760.521,E2 5760.521} C_VEL
LIN {X 0,Y 324.503,Z 733.224,A -85,B 0,C 180,E1 5760.179,E2 5760.179} C_VEL
LIN {X 0,Y 319.452,Z 756.207,A -85,B 0,C 180,E1 5759.846,E2 5759.846} C_VEL
LIN {X 0,Y 312.66,Z 778.827,A -85,B 0,C 180,E1 5759.477,E2 5759.477} C_VEL
LIN {X 0,Y 304.47,Z 800.825,A -85,B 0,C 180,E1 5759.011,E2 5759.011} C_VEL
LIN {X 0,Y 295.038,Z 821.422,A -85,B 0,C 180,E1 5758.427,E2 5758.427} C_VEL
LIN {X 0,Y 293.03,Z 825.52,A -85,B 0,C 180,E1 5758.289,E2 5758.289} C_VEL
LIN {X 0,Y 289.452,Z 832.411,A -85,B 0,C 180,E1 5758.241,E2 5758.241} C_VEL
LIN {X 0,Y 279.175,Z 849.504,A -85,B 0,C 180,E1 5758.781,E2 5758.781} C_VEL
LIN {X 0,Y 274.919,Z 855.959,A -85,B 0,C 180,E1 5758.697,E2 5758.697} C_VEL
LIN {X 0,Y 262.633,Z 873.507,A -85,B 0,C 180,E1 5757.777,E2 5757.777} C_VEL
LIN {X 0,Y 247.406,Z 892.516,A -85,B 0,C 180,E1 5756.479,E2 5756.479} C_VEL
LIN {X 0,Y 232.331,Z 909.059,A -85,B 0,C 180,E1 5754.99,E2 5754.99} C_VEL
LIN {X 0,Y 215.535,Z 925.234,A -85,B 0,C 180,E1 5753.043,E2 5753.043} C_VEL
LIN {X 0,Y 198.574,Z 939.816,A -85,B 0,C 180,E1 5750.679,E2 5750.679} C_VEL
LIN {X 0,Y 181.112,Z 952.975,A -85,B 0,C 180,E1 5747.704,E2 5747.704} C_VEL
LIN {X 0,Y 163.376,Z 965.032,A -85,B 0,C 180,E1 5743.892,E2 5743.892} C_VEL
LIN {X 0,Y 145.707,Z 975.629,A -85,B 0,C 180,E1 5738.932,E2 5738.932} C_VEL
LIN {X 0,Y 127.916,Z 985.294,A -85,B 0,C 180,E1 5732.029,E2 5732.029} C_VEL
LIN {X 0,Y 113.653,Z 992.413,A -85,B 0,C 180,E1 5724.028,E2 5724.028} C_VEL
LIN {X 0,Y 100.7,Z 998.587,A -85,B 0,C 180,E1 5712.716,E2 5712.716} C_VEL
LIN {X 0,Y 92.646,Z 1002.668,A -85,B 0,C 180,E1 5700.305,E2 5700.305} C_VEL
LIN {X 0,Y 88.648,Z 1005.196,A -85,B 0,C 180,E1 5686.378,E2 5686.378} C_VEL
LIN {X 0,Y 88.06,Z 1006.107,A -85,B 0,C 180,E1 5675.866,E2 5675.866} C_VEL
LIN {X 0,Y 88.091,Z 1006.255,A -85,B 0,C 180,E1 5668.051,E2 5668.051} C_VEL
LIN {X 0,Y 88.156,Z 1005.783,A -85,B 0,C 180,E1 5658.886,E2 5658.886} C_VEL
LIN {X 0,Y 90.154,Z 1004.061,A -85,B 0,C 180,E1 5646.473,E2 5646.473} C_VEL
LIN {X 0,Y 95.97,Z 1000.9,A -85,B 0,C 180,E1 5633.576,E2 5633.576} C_VEL
LIN {X 0,Y 106.606,Z 995.721,A -85,B 0,C 180,E1 5621.392,E2 5621.392} C_VEL
LIN {X 0,Y 120.848,Z 988.878,A -85,B 0,C 180,E1 5611.563,E2 5611.563} C_VEL
LIN {X 0,Y 137.045,Z 980.368,A -85,B 0,C 180,E1 5604.114,E2 5604.114} C_VEL
LIN {X 0,Y 154.814,Z 970.207,A -85,B 0,C 180,E1 5598.329,E2 5598.329} C_VEL
LIN {X 0,Y 172.137,Z 959.107,A -85,B 0,C 180,E1 5594.095,E2 5594.095} C_VEL
LIN {X 0,Y 191.147,Z 945.403,A -85,B 0,C 180,E1 5590.495,E2 5590.495} C_VEL
LIN {X 0,Y 208.889,Z 931.038,A -85,B 0,C 180,E1 5587.825,E2 5587.825} C_VEL
LIN {X 0,Y 226.054,Z 915.103,A -85,B 0,C 180,E1 5585.692,E2 5585.692} C_VEL
LIN {X 0,Y 242.518,Z 897.878,A -85,B 0,C 180,E1 5583.974,E2 5583.974} C_VEL
LIN {X 0,Y 256.224,Z 881.532,A -85,B 0,C 180,E1 5582.737,E2 5582.737} C_VEL
LIN {X 0,Y 271.029,Z 861.408,A -85,B 0,C 180,E1 5581.57,E2 5581.57} C_VEL
LIN {X 0,Y 282.948,Z 842.703,A -85,B 0,C 180,E1 5580.737,E2 5580.737} C_VEL
LIN {X 0,Y 294.711,Z 821.075,A -85,B 0,C 180,E1 5580,E2 5580} C_VEL
LIN {X 0,Y 301.328,Z 807.022,A -85,B 0,C 180,E1 5579.619,E2 5579.619} C_VEL
LIN {X 0,Y 290.977,Z 828.264,A -85,B 0,C 180,E1 5578.892,E2 5578.892} C_VEL
LIN {X 0,Y 280.082,Z 847.073,A -85,B 0,C 180,E1 5578.083,E2 5578.083} C_VEL
LIN {X 0,Y 266.304,Z 867.599,A -85,B 0,C 180,E1 5576.96,E2 5576.96} C_VEL
LIN {X 0,Y 253.122,Z 884.616,A -85,B 0,C 180,E1 5575.769,E2 5575.769} C_VEL
LIN {X 0,Y 237.174,Z 902.591,A -85,B 0,C 180,E1 5574.145,E2 5574.145} C_VEL
LIN {X 0,Y 220.967,Z 918.678,A -85,B 0,C 180,E1 5572.236,E2 5572.236} C_VEL
LIN {X 0,Y 204.104,Z 933.235,A -85,B 0,C 180,E1 5569.907,E2 5569.907} C_VEL
LIN {X 0,Y 186.715,Z 946.645,A -85,B 0,C 180,E1 5567.002,E2 5567.002} C_VEL
LIN {X 0,Y 169.039,Z 958.565,A -85,B 0,C 180,E1 5563.355,E2 5563.355} C_VEL
LIN {X 0,Y 150.513,Z 969.65,A -85,B 0,C 180,E1 5558.418,E2 5558.418} C_VEL
LIN {X 0,Y 134.08,Z 978.408,A -85,B 0,C 180,E1 5552.534,E2 5552.534} C_VEL
LIN {X 0,Y 118.636,Z 985.76,A -85,B 0,C 180,E1 5544.824,E2 5544.824} C_VEL
LIN {X 0,Y 105.164,Z 991.781,A -85,B 0,C 180,E1 5534.705,E2 5534.705} C_VEL
LIN {X 0,Y 95.284,Z 995.934,A -85,B 0,C 180,E1 5522.349,E2 5522.349} C_VEL
LIN {X 0,Y 89.873,Z 998.528,A -85,B 0,C 180,E1 5508.818,E2 5508.818} C_VEL
LIN {X 0,Y 88.265,Z 999.487,A -85,B 0,C 180,E1 5497.155,E2 5497.155} C_VEL
LIN {X 0,Y 88.122,Z 999.657,A -85,B 0,C 180,E1 5488.048,E2 5488.048} C_VEL
LIN {X 0,Y 88.714,Z 999.17,A -85,B 0,C 180,E1 5477.635,E2 5477.635} C_VEL
LIN {X 0,Y 91.564,Z 997.638,A -85,B 0,C 180,E1 5465.485,E2 5465.485} C_VEL
LIN {X 0,Y 98.626,Z 994.608,A -85,B 0,C 180,E1 5452.538,E2 5452.538} C_VEL
LIN {X 0,Y 109.425,Z 989.911,A -85,B 0,C 180,E1 5441.478,E2 5441.478} C_VEL
LIN {X 0,Y 123.939,Z 983.416,A -85,B 0,C 180,E1 5432.114,E2 5432.114} C_VEL
LIN {X 0,Y 139.333,Z 975.774,A -85,B 0,C 180,E1 5425.298,E2 5425.298} C_VEL
LIN {X 0,Y 157.898,Z 965.505,A -85,B 0,C 180,E1 5419.365,E2 5419.365} C_VEL
LIN {X 0,Y 175.099,Z 954.796,A -85,B 0,C 180,E1 5415.217,E2 5415.217} C_VEL
LIN {X 0,Y 193.029,Z 942.082,A -85,B 0,C 180,E1 5411.794,E2 5411.794} C_VEL
LIN {X 0,Y 210.587,Z 928.099,A -85,B 0,C 180,E1 5409.077,E2 5409.077} C_VEL
LIN {X 0,Y 226.628,Z 913.448,A -85,B 0,C 180,E1 5406.986,E2 5406.986} C_VEL
LIN {X 0,Y 242.93,Z 896.69,A -85,B 0,C 180,E1 5405.172,E2 5405.172} C_VEL
LIN {X 0,Y 257.006,Z 880.113,A -85,B 0,C 180,E1 5403.793,E2 5403.793} C_VEL
LIN {X 0,Y 271.442,Z 860.68,A -85,B 0,C 180,E1 5402.534,E2 5402.534} C_VEL
LIN {X 0,Y 283.042,Z 842.659,A -85,B 0,C 180,E1 5401.613,E2 5401.613} C_VEL
LIN {X 0,Y 294.433,Z 822.025,A -85,B 0,C 180,E1 5400.779,E2 5400.779} C_VEL
LIN {X 0,Y 300.806,Z 808.761,A -85,B 0,C 180,E1 5400.331,E2 5400.331} C_VEL
LIN {X 0,Y 289.932,Z 830.76,A -85,B 0,C 180,E1 5399.694,E2 5399.694} C_VEL
LIN {X 0,Y 278.818,Z 849.883,A -85,B 0,C 180,E1 5398.973,E2 5398.973} C_VEL
LIN {X 0,Y 274.919,Z 855.959,A -85,B 0,C 180,E1 5398.697,E2 5398.697} C_VEL
LIN {X 0,Y 270.512,Z 862.487,A -85,B 0,C 180,E1 5398.596,E2 5398.596} C_VEL
LIN {X 0,Y 258.485,Z 878.485,A -85,B 0,C 180,E1 5399.049,E2 5399.049} C_VEL
LIN {X 0,Y 253.662,Z 884.359,A -85,B 0,C 180,E1 5398.914,E2 5398.914} C_VEL
LIN {X 0,Y 237.162,Z 903.112,A -85,B 0,C 180,E1 5397.531,E2 5397.531} C_VEL
LIN {X 0,Y 221.489,Z 918.75,A -85,B 0,C 180,E1 5395.988,E2 5395.988} C_VEL
LIN {X 0,Y 204.083,Z 934.027,A -85,B 0,C 180,E1 5393.961,E2 5393.961} C_VEL
LIN {X 0,Y 186.99,Z 947.376,A -85,B 0,C 180,E1 5391.54,E2 5391.54} C_VEL
LIN {X 0,Y 168.476,Z 960.078,A -85,B 0,C 180,E1 5388.274,E2 5388.274} C_VEL
LIN {X 0,Y 149.779,Z 971.546,A -85,B 0,C 180,E1 5383.985,E2 5383.985} C_VEL
LIN {X 0,Y 132.117,Z 981.017,A -85,B 0,C 180,E1 5378.556,E2 5378.556} C_VEL
LIN {X 0,Y 114.511,Z 989.581,A -85,B 0,C 180,E1 5370.818,E2 5370.818} C_VEL
LIN {X 0,Y 100.681,Z 995.719,A -85,B 0,C 180,E1 5361.673,E2 5361.673} C_VEL
LIN {X 0,Y 88.603,Z 1000.958,A -85,B 0,C 180,E1 5348.361,E2 5348.361} C_VEL
LIN {X 0,Y 82.471,Z 1003.896,A -85,B 0,C 180,E1 5335.108,E2 5335.108} C_VEL
LIN {X 0,Y 80.142,Z 1005.632,A -85,B 0,C 180,E1 5320.787,E2 5320.787} C_VEL
LIN {X 0,Y 80.108,Z 1006.007,A -85,B 0,C 180,E1 5310.717,E2 5310.717} C_VEL
LIN {X 0,Y 80.083,Z 1005.719,A -85,B 0,C 180,E1 5301.386,E2 5301.386} C_VEL
LIN {X 0,Y 81.876,Z 1004.242,A -85,B 0,C 180,E1 5287.002,E2 5287.002} C_VEL
LIN {X 0,Y 87.883,Z 1001.24,A -85,B 0,C 180,E1 5272.785,E2 5272.785} C_VEL
LIN {X 0,Y 98.919,Z 996.469,A -85,B 0,C 180,E1 5259.819,E2 5259.819} C_VEL
LIN {X 0,Y 113.079,Z 990.152,A -85,B 0,C 180,E1 5249.956,E2 5249.956} C_VEL
LIN {X 0,Y 131.302,Z 981.354,A -85,B 0,C 180,E1 5241.737,E2 5241.737} C_VEL
LIN {X 0,Y 148.902,Z 971.929,A -85,B 0,C 180,E1 5236.24,E2 5236.24} C_VEL
LIN {X 0,Y 167.559,Z 960.549,A -85,B 0,C 180,E1 5231.904,E2 5231.904} C_VEL
LIN {X 0,Y 186.043,Z 947.941,A -85,B 0,C 180,E1 5228.602,E2 5228.602} C_VEL
LIN {X 0,Y 203.116,Z 934.64,A -85,B 0,C 180,E1 5226.154,E2 5226.154} C_VEL
LIN {X 0,Y 220.507,Z 919.48,A -85,B 0,C 180,E1 5224.107,E2 5224.107} C_VEL
LIN {X 0,Y 236.44,Z 903.625,A -85,B 0,C 180,E1 5222.525,E2 5222.525} C_VEL
LIN {X 0,Y 252.981,Z 884.906,A -85,B 0,C 180,E1 5221.128,E2 5221.128} C_VEL
LIN {X 0,Y 266.929,Z 866.82,A -85,B 0,C 180,E1 5220.109,E2 5220.109} C_VEL
LIN {X 0,Y 276.5,Z 852.858,A -85,B 0,C 180,E1 5219.484,E2 5219.484} C_VEL
LIN {X 0,Y 263.518,Z 871.214,A -85,B 0,C 180,E1 5218.509,E2 5218.509} C_VEL
LIN {X 0,Y 248.38,Z 889.952,A -85,B 0,C 180,E1 5217.231,E2 5217.231} C_VEL
LIN {X 0,Y 233.559,Z 905.903,A -85,B 0,C 180,E1 5215.819,E2 5215.819} C_VEL
LIN {X 0,Y 216.077,Z 922.428,A -85,B 0,C 180,E1 5213.89,E2 5213.89} C_VEL
LIN {X 0,Y 199.994,Z 935.819,A -85,B 0,C 180,E1 5211.795,E2 5211.795} C_VEL
LIN {X 0,Y 181.367,Z 949.435,A -85,B 0,C 180,E1 5208.863,E2 5208.863} C_VEL
LIN {X 0,Y 163.303,Z 961.121,A -85,B 0,C 180,E1 5205.298,E2 5205.298} C_VEL
LIN {X 0,Y 145.137,Z 971.302,A -85,B 0,C 180,E1 5200.678,E2 5200.678} C_VEL
LIN {X 0,Y 127.347,Z 980.201,A -85,B 0,C 180,E1 5194.528,E2 5194.528} C_VEL
LIN {X 0,Y 111.874,Z 987.002,A -85,B 0,C 180,E1 5186.962,E2 5186.962} C_VEL
LIN {X 0,Y 96.729,Z 993.082,A -85,B 0,C 180,E1 5175.49,E2 5175.49} C_VEL
LIN {X 0,Y 87.362,Z 996.694,A -85,B 0,C 180,E1 5163.317,E2 5163.317} C_VEL
LIN {X 0,Y 81.569,Z 999.079,A -85,B 0,C 180,E1 5147.841,E2 5147.841} C_VEL
LIN {X 0,Y 80.231,Z 999.827,A -85,B 0,C 180,E1 5136.437,E2 5136.437} C_VEL
LIN {X 0,Y 80.131,Z 999.936,A -85,B 0,C 180,E1 5127.137,E2 5127.137} C_VEL
LIN {X 0,Y 80.936,Z 999.41,A -85,B 0,C 180,E1 5115.695,E2 5115.695} C_VEL
LIN {X 0,Y 84.416,Z 997.862,A -85,B 0,C 180,E1 5102.668,E2 5102.668} C_VEL
LIN {X 0,Y 93.169,Z 994.522,A -85,B 0,C 180,E1 5088.294,E2 5088.294} C_VEL
LIN {X 0,Y 104.755,Z 989.976,A -85,B 0,C 180,E1 5077.613,E2 5077.613} C_VEL
LIN {X 0,Y 121.264,Z 983.02,A -85,B 0,C 180,E1 5068.034,E2 5068.034} C_VEL
LIN {X 0,Y 137.627,Z 975.296,A -85,B 0,C 180,E1 5061.592,E2 5061.592} C_VEL
LIN {X 0,Y 156.22,Z 965.311,A -85,B 0,C 180,E1 5056.269,E2 5056.269} C_VEL
LIN {X 0,Y 174.023,Z 954.542,A -85,B 0,C 180,E1 5052.406,E2 5052.406} C_VEL
LIN {X 0,Y 192.161,Z 941.913,A -85,B 0,C 180,E1 5049.283,E2 5049.283} C_VEL
LIN {X 0,Y 209.505,Z 928.354,A -85,B 0,C 180,E1 5046.853,E2 5046.853} C_VEL
LIN {X 0,Y 225.779,Z 913.751,A -85,B 0,C 180,E1 5044.926,E2 5044.926} C_VEL
LIN {X 0,Y 242.331,Z 896.992,A -85,B 0,C 180,E1 5043.252,E2 5043.252} C_VEL
LIN {X 0,Y 256.224,Z 880.868,A -85,B 0,C 180,E1 5042.013,E2 5042.013} C_VEL
LIN {X 0,Y 270.962,Z 861.333,A -85,B 0,C 180,E1 5040.843,E2 5040.843} C_VEL
LIN {X 0,Y 275.941,Z 854.052,A -85,B 0,C 180,E1 5040.467,E2 5040.467} C_VEL
LIN {X 0,Y 262.941,Z 872.531,A -85,B 0,C 180,E1 5039.602,E2 5039.602} C_VEL
LIN {X 0,Y 253.662,Z 884.359,A -85,B 0,C 180,E1 5038.914,E2 5038.914} C_VEL
LIN {X 0,Y 248.677,Z 890.301,A -85,B 0,C 180,E1 5038.759,E2 5038.759} C_VEL
LIN {X 0,Y 235,Z 904.972,A -85,B 0,C 180,E1 5039.114,E2 5039.114} C_VEL
LIN {X 0,Y 229.547,Z 910.41,A -85,B 0,C 180,E1 5038.901,E2 5038.901} C_VEL
LIN {X 0,Y 212.192,Z 926.332,A -85,B 0,C 180,E1 5037.252,E2 5037.252} C_VEL
LIN {X 0,Y 193.657,Z 941.364,A -85,B 0,C 180,E1 5035.114,E2 5035.114} C_VEL
LIN {X 0,Y 176.401,Z 953.647,A -85,B 0,C 180,E1 5032.665,E2 5032.665} C_VEL
LIN {X 0,Y 155.614,Z 966.656,A -85,B 0,C 180,E1 5028.887,E2 5028.887} C_VEL
LIN {X 0,Y 136.871,Z 976.978,A -85,B 0,C 180,E1 5024.32,E2 5024.32} C_VEL
LIN {X 0,Y 118.52,Z 985.763,A -85,B 0,C 180,E1 5018.11,E2 5018.11} C_VEL
LIN {X 0,Y 101.826,Z 993.013,A -85,B 0,C 180,E1 5009.772,E2 5009.772} C_VEL
LIN {X 0,Y 87.851,Z 998.469,A -85,B 0,C 180,E1 4998.686,E2 4998.686} C_VEL
LIN {X 0,Y 77.459,Z 1002.603,A -85,B 0,C 180,E1 4983.713,E2 4983.713} C_VEL
LIN {X 0,Y 72.864,Z 1004.736,A -85,B 0,C 180,E1 4968.398,E2 4968.398} C_VEL
LIN {X 0,Y 72.066,Z 1005.53,A -85,B 0,C 180,E1 4956.374,E2 4956.374} C_VEL
LIN {X 0,Y 72.091,Z 1005.655,A -85,B 0,C 180,E1 4947.618,E2 4947.618} C_VEL
LIN {X 0,Y 72.301,Z 1005.174,A -85,B 0,C 180,E1 4936.407,E2 4936.407} C_VEL
LIN {X 0,Y 75.594,Z 1003.334,A -85,B 0,C 180,E1 4920.801,E2 4920.801} C_VEL
LIN {X 0,Y 84.254,Z 999.902,A -85,B 0,C 180,E1 4905.398,E2 4905.398} C_VEL
LIN {X 0,Y 97.692,Z 994.56,A -85,B 0,C 180,E1 4892.951,E2 4892.951} C_VEL
LIN {X 0,Y 114.532,Z 987.517,A -85,B 0,C 180,E1 4883.579,E2 4883.579} C_VEL
LIN {X 0,Y 131.84,Z 979.369,A -85,B 0,C 180,E1 4877.169,E2 4877.169} C_VEL
LIN {X 0,Y 152.197,Z 968.52,A -85,B 0,C 180,E1 4871.84,E2 4871.84} C_VEL
LIN {X 0,Y 170.724,Z 957.304,A -85,B 0,C 180,E1 4868.258,E2 4868.258} C_VEL
LIN {X 0,Y 189.786,Z 944.06,A -85,B 0,C 180,E1 4865.385,E2 4865.385} C_VEL
LIN {X 0,Y 208.261,Z 929.57,A -85,B 0,C 180,E1 4863.163,E2 4863.163} C_VEL
LIN {X 0,Y 225.016,Z 914.477,A -85,B 0,C 180,E1 4861.493,E2 4861.493} C_VEL
LIN {X 0,Y 241.935,Z 897.253,A -85,B 0,C 180,E1 4860.078,E2 4860.078} C_VEL
LIN {X 0,Y 251.451,Z 886.433,A -85,B 0,C 180,E1 4859.373,E2 4859.373} C_VEL
LIN {X 0,Y 235.69,Z 903.593,A -85,B 0,C 180,E1 4858.055,E2 4858.055} C_VEL
LIN {X 0,Y 219.355,Z 919.297,A -85,B 0,C 180,E1 4856.477,E2 4856.477} C_VEL
LIN {X 0,Y 201.874,Z 933.856,A -85,B 0,C 180,E1 4854.501,E2 4854.501} C_VEL
LIN {X 0,Y 183.73,Z 947.255,A -85,B 0,C 180,E1 4852.02,E2 4852.02} C_VEL
LIN {X 0,Y 165.068,Z 959.188,A -85,B 0,C 180,E1 4848.856,E2 4848.856} C_VEL
LIN {X 0,Y 144.748,Z 970.526,A -85,B 0,C 180,E1 4844.371,E2 4844.371} C_VEL
LIN {X 0,Y 126.469,Z 979.425,A -85,B 0,C 180,E1 4838.871,E2 4838.871} C_VEL
LIN {X 0,Y 109.196,Z 986.674,A -85,B 0,C 180,E1 4831.51,E2 4831.51} C_VEL
LIN {X 0,Y 93.543,Z 992.606,A -85,B 0,C 180,E1 4821.275,E2 4821.275} C_VEL
LIN {X 0,Y 81.905,Z 996.55,A -85,B 0,C 180,E1 4808.497,E2 4808.497} C_VEL
LIN {X 0,Y 74.687,Z 999.137,A -85,B 0,C 180,E1 4792.839,E2 4792.839} C_VEL
LIN {X 0,Y 72.357,Z 1000.089,A -85,B 0,C 180,E1 4778.74,E2 4778.74} C_VEL
LIN {X 0,Y 72.134,Z 1000.257,A -85,B 0,C 180,E1 4767.615,E2 4767.615} C_VEL
LIN {X 0,Y 73.01,Z 999.775,A -85,B 0,C 180,E1 4754.918,E2 4754.918} C_VEL
LIN {X 0,Y 77.019,Z 998.248,A -85,B 0,C 180,E1 4740.438,E2 4740.438} C_VEL
LIN {X 0,Y 86.155,Z 995.223,A -85,B 0,C 180,E1 4725.872,E2 4725.872} C_VEL
LIN {X 0,Y 99.254,Z 990.529,A -85,B 0,C 180,E1 4714.312,E2 4714.312} C_VEL
LIN {X 0,Y 115.988,Z 984.034,A -85,B 0,C 180,E1 4705.17,E2 4705.17} C_VEL
LIN {X 0,Y 133.1,Z 976.393,A -85,B 0,C 180,E1 4698.838,E2 4698.838} C_VEL
LIN {X 0,Y 153.208,Z 966.123,A -85,B 0,C 180,E1 4693.517,E2 4693.517} C_VEL
LIN {X 0,Y 171.507,Z 955.411,A -85,B 0,C 180,E1 4689.888,E2 4689.888} C_VEL
LIN {X 0,Y 190.348,Z 942.695,A -85,B 0,C 180,E1 4686.937,E2 4686.937} C_VEL
LIN {X 0,Y 208.628,Z 928.709,A -85,B 0,C 180,E1 4684.622,E2 4684.622} C_VEL
LIN {X 0,Y 225.224,Z 914.055,A -85,B 0,C 180,E1 4682.853,E2 4682.853} C_VEL
LIN {X 0,Y 242.005,Z 897.294,A -85,B 0,C 180,E1 4681.325,E2 4681.325} C_VEL
LIN {X 0,Y 250.951,Z 887.345,A -85,B 0,C 180,E1 4680.58,E2 4680.58} C_VEL
LIN {X 0,Y 234.957,Z 904.856,A -85,B 0,C 180,E1 4679.362,E2 4679.362} C_VEL
LIN {X 0,Y 229.547,Z 910.41,A -85,B 0,C 180,E1 4678.901,E2 4678.901} C_VEL
LIN {X 0,Y 223.952,Z 915.715,A -85,B 0,C 180,E1 4678.663,E2 4678.663} C_VEL
LIN {X 0,Y 207.856,Z 929.596,A -85,B 0,C 180,E1 4678.886,E2 4678.886} C_VEL
LIN {X 0,Y 202.725,Z 933.632,A -85,B 0,C 180,E1 4678.601,E2 4678.601} C_VEL
LIN {X 0,Y 184.294,Z 947.468,A -85,B 0,C 180,E1 4676.526,E2 4676.526} C_VEL
LIN {X 0,Y 164.928,Z 960.04,A -85,B 0,C 180,E1 4673.793,E2 4673.793} C_VEL
LIN {X 0,Y 145.113,Z 971.391,A -85,B 0,C 180,E1 4670.132,E2 4670.132} C_VEL
LIN {X 0,Y 126.061,Z 980.807,A -85,B 0,C 180,E1 4665.366,E2 4665.366} C_VEL
LIN {X 0,Y 105.714,Z 989.583,A -85,B 0,C 180,E1 4657.943,E2 4657.943} C_VEL
LIN {X 0,Y 89.152,Z 995.891,A -85,B 0,C 180,E1 4648.461,E2 4648.461} C_VEL
LIN {X 0,Y 75.243,Z 1000.676,A -85,B 0,C 180,E1 4634.768,E2 4634.768} C_VEL
LIN {X 0,Y 67.024,Z 1003.669,A -85,B 0,C 180,E1 4618.344,E2 4618.344} C_VEL
LIN {X 0,Y 64.144,Z 1005.117,A -85,B 0,C 180,E1 4600.782,E2 4600.782} C_VEL
LIN {X 0,Y 64.127,Z 1005.422,A -85,B 0,C 180,E1 4590.002,E2 4590.002} C_VEL
LIN {X 0,Y 64.148,Z 1005.108,A -85,B 0,C 180,E1 4579.091,E2 4579.091} C_VEL
LIN {X 0,Y 67.068,Z 1003.625,A -85,B 0,C 180,E1 4561.513,E2 4561.513} C_VEL
LIN {X 0,Y 75.239,Z 1000.645,A -85,B 0,C 180,E1 4545.235,E2 4545.235} C_VEL
LIN {X 0,Y 89.147,Z 995.841,A -85,B 0,C 180,E1 4531.54,E2 4531.54} C_VEL
LIN {X 0,Y 105.708,Z 989.521,A -85,B 0,C 180,E1 4522.055,E2 4522.055} C_VEL
LIN {X 0,Y 126.054,Z 980.722,A -85,B 0,C 180,E1 4514.631,E2 4514.631} C_VEL
LIN {X 0,Y 145.105,Z 971.297,A -85,B 0,C 180,E1 4509.864,E2 4509.864} C_VEL
LIN {X 0,Y 164.92,Z 959.917,A -85,B 0,C 180,E1 4506.202,E2 4506.202} C_VEL
LIN {X 0,Y 184.287,Z 947.311,A -85,B 0,C 180,E1 4503.467,E2 4503.467} C_VEL
LIN {X 0,Y 202.487,Z 933.637,A -85,B 0,C 180,E1 4501.414,E2 4501.414} C_VEL
LIN {X 0,Y 220.943,Z 917.915,A -85,B 0,C 180,E1 4499.717,E2 4499.717} C_VEL
LIN {X 0,Y 226.353,Z 912.854,A -85,B 0,C 180,E1 4499.273,E2 4499.273} C_VEL
LIN {X 0,Y 210.104,Z 927.134,A -85,B 0,C 180,E1 4497.757,E2 4497.757} C_VEL
LIN {X 0,Y 191.488,Z 941.443,A -85,B 0,C 180,E1 4495.694,E2 4495.694} C_VEL
LIN {X 0,Y 173.168,Z 953.794,A -85,B 0,C 180,E1 4493.209,E2 4493.209} C_VEL
LIN {X 0,Y 153.715,Z 965.107,A -85,B 0,C 180,E1 4489.884,E2 4489.884} C_VEL
LIN {X 0,Y 134.249,Z 975.017,A -85,B 0,C 180,E1 4485.484,E2 4485.484} C_VEL
LIN {X 0,Y 115.243,Z 983.217,A -85,B 0,C 180,E1 4479.535,E2 4479.535} C_VEL
LIN {X 0,Y 96.346,Z 990.278,A -85,B 0,C 180,E1 4470.646,E2 4470.646} C_VEL
LIN {X 0,Y 82.027,Z 994.954,A -85,B 0,C 180,E1 4459.755,E2 4459.755} C_VEL
LIN {X 0,Y 70.432,Z 998.415,A -85,B 0,C 180,E1 4443.611,E2 4443.611} C_VEL
LIN {X 0,Y 65.394,Z 999.996,A -85,B 0,C 180,E1 4427.801,E2 4427.801} C_VEL
LIN {X 0,Y 64.16,Z 1000.516,A -85,B 0,C 180,E1 4414.13,E2 4414.13} C_VEL
LIN {X 0,Y 64.22,Z 1000.475,A -85,B 0,C 180,E1 4403.741,E2 4403.741} C_VEL
LIN {X 0,Y 65.713,Z 999.892,A -85,B 0,C 180,E1 4390.443,E2 4390.443} C_VEL
LIN {X 0,Y 71.501,Z 998.151,A -85,B 0,C 180,E1 4374.202,E2 4374.202} C_VEL
LIN {X 0,Y 83.418,Z 994.548,A -85,B 0,C 180,E1 4358.828,E2 4358.828} C_VEL
LIN {X 0,Y 98.53,Z 989.619,A -85,B 0,C 180,E1 4348.02,E2 4348.02} C_VEL
LIN {X 0,Y 116.034,Z 982.976,A -85,B 0,C 180,E1 4340.089,E2 4340.089} C_VEL
LIN {X 0,Y 135.104,Z 974.725,A -85,B 0,C 180,E1 4334.211,E2 4334.211} C_VEL
LIN {X 0,Y 154.273,Z 964.922,A -85,B 0,C 180,E1 4329.926,E2 4329.926} C_VEL
LIN {X 0,Y 174.102,Z 953.335,A -85,B 0,C 180,E1 4326.57,E2 4326.57} C_VEL
LIN {X 0,Y 191.821,Z 941.38,A -85,B 0,C 180,E1 4324.186,E2 4324.186} C_VEL
LIN {X 0,Y 211.086,Z 926.516,A -85,B 0,C 180,E1 4322.065,E2 4322.065} C_VEL
LIN {X 0,Y 225.912,Z 913.491,A -85,B 0,C 180,E1 4320.682,E2 4320.682} C_VEL
LIN {X 0,Y 208.613,Z 928.903,A -85,B 0,C 180,E1 4319.177,E2 4319.177} C_VEL
LIN {X 0,Y 202.725,Z 933.632,A -85,B 0,C 180,E1 4318.601,E2 4318.601} C_VEL
LIN {X 0,Y 196.61,Z 938.42,A -85,B 0,C 180,E1 4318.271,E2 4318.271} C_VEL
LIN {X 0,Y 180.057,Z 949.822,A -85,B 0,C 180,E1 4318.361,E2 4318.361} C_VEL
LIN {X 0,Y 173.678,Z 953.926,A -85,B 0,C 180,E1 4317.93,E2 4317.93} C_VEL
LIN {X 0,Y 153.528,Z 965.89,A -85,B 0,C 180,E1 4315.086,E2 4315.086} C_VEL
LIN {X 0,Y 133.497,Z 976.261,A -85,B 0,C 180,E1 4311.322,E2 4311.322} C_VEL
LIN {X 0,Y 113.336,Z 985.135,A -85,B 0,C 180,E1 4306.01,E2 4306.01} C_VEL
LIN {X 0,Y 94.502,Z 992.386,A -85,B 0,C 180,E1 4298.588,E2 4298.588} C_VEL
LIN {X 0,Y 77.845,Z 997.844,A -85,B 0,C 180,E1 4287.957,E2 4287.957} C_VEL
LIN {X 0,Y 64.181,Z 1002.03,A -85,B 0,C 180,E1 4271.605,E2 4271.605} C_VEL
LIN {X 0,Y 57.581,Z 1004.123,A -85,B 0,C 180,E1 4253.539,E2 4253.539} C_VEL
LIN {X 0,Y 56.07,Z 1004.954,A -85,B 0,C 180,E1 4237.173,E2 4237.173} C_VEL
LIN {X 0,Y 56.103,Z 1005.079,A -85,B 0,C 180,E1 4227.96,E2 4227.96} C_VEL
LIN {X 0,Y 56.513,Z 1004.639,A -85,B 0,C 180,E1 4213.561,E2 4213.561} C_VEL
LIN {X 0,Y 61.369,Z 1002.824,A -85,B 0,C 180,E1 4194.096,E2 4194.096} C_VEL
LIN {X 0,Y 71.972,Z 999.651,A -85,B 0,C 180,E1 4177.652,E2 4177.652} C_VEL
LIN {X 0,Y 88.181,Z 994.444,A -85,B 0,C 180,E1 4164.803,E2 4164.803} C_VEL
LIN {X 0,Y 107.161,Z 987.614,A -85,B 0,C 180,E1 4156.075,E2 4156.075} C_VEL
LIN {X 0,Y 126.966,Z 979.154,A -85,B 0,C 180,E1 4150.186,E2 4150.186} C_VEL
LIN {X 0,Y 148.125,Z 968.729,A -85,B 0,C 180,E1 4145.81,E2 4145.81} C_VEL
LIN {X 0,Y 167.169,Z 957.845,A -85,B 0,C 180,E1 4142.902,E2 4142.902} C_VEL
LIN {X 0,Y 187.955,Z 944.143,A -85,B 0,C 180,E1 4140.448,E2 4140.448} C_VEL
LIN {X 0,Y 200.967,Z 934.477,A -85,B 0,C 180,E1 4139.165,E2 4139.165} C_VEL
LIN {X 0,Y 182.175,Z 947.876,A -85,B 0,C 180,E1 4137.155,E2 4137.155} C_VEL
LIN {X 0,Y 162.685,Z 959.811,A -85,B 0,C 180,E1 4134.573,E2 4134.573} C_VEL
LIN {X 0,Y 141.724,Z 970.896,A -85,B 0,C 180,E1 4130.953,E2 4130.953} C_VEL
LIN {X 0,Y 122.384,Z 979.656,A -85,B 0,C 180,E1 4126.429,E2 4126.429} C_VEL
LIN {X 0,Y 103.18,Z 987.005,A -85,B 0,C 180,E1 4120.025,E2 4120.025} C_VEL
LIN {X 0,Y 84.945,Z 993.021,A -85,B 0,C 180,E1 4110.563,E2 4110.563} C_VEL
LIN {X 0,Y 69.815,Z 997.166,A -85,B 0,C 180,E1 4096.91,E2 4096.91} C_VEL
LIN {X 0,Y 59.724,Z 999.808,A -85,B 0,C 180,E1 4077.947,E2 4077.947} C_VEL
LIN {X 0,Y 56.438,Z 1000.711,A -85,B 0,C 180,E1 4060.2,E2 4060.2} C_VEL
LIN {X 0,Y 56.148,Z 1000.857,A -85,B 0,C 180,E1 4046.935,E2 4046.935} C_VEL
LIN {X 0,Y 57.542,Z 1000.382,A -85,B 0,C 180,E1 4030.722,E2 4030.722} C_VEL
LIN {X 0,Y 63.327,Z 998.86,A -85,B 0,C 180,E1 4013.134,E2 4013.134} C_VEL
LIN {X 0,Y 75.857,Z 995.643,A -85,B 0,C 180,E1 3996.489,E2 3996.489} C_VEL
LIN {X 0,Y 91.748,Z 990.903,A -85,B 0,C 180,E1 3985.251,E2 3985.251} C_VEL
LIN {X 0,Y 111.709,Z 983.969,A -85,B 0,C 180,E1 3976.739,E2 3976.739} C_VEL
LIN {X 0,Y 130.546,Z 976.224,A -85,B 0,C 180,E1 3971.402,E2 3971.402} C_VEL
LIN {X 0,Y 151.158,Z 966.237,A -85,B 0,C 180,E1 3967.204,E2 3967.204} C_VEL
LIN {X 0,Y 170.428,Z 955.465,A -85,B 0,C 180,E1 3964.252,E2 3964.252} C_VEL
LIN {X 0,Y 189.067,Z 943.307,A -85,B 0,C 180,E1 3961.981,E2 3961.981} C_VEL
LIN {X 0,Y 200.745,Z 934.84,A -85,B 0,C 180,E1 3960.777,E2 3960.777} C_VEL
LIN {X 0,Y 181.989,Z 948.494,A -85,B 0,C 180,E1 3958.902,E2 3958.902} C_VEL
LIN {X 0,Y 173.678,Z 953.926,A -85,B 0,C 180,E1 3957.93,E2 3957.93} C_VEL
LIN {X 0,Y 167.201,Z 957.978,A -85,B 0,C 180,E1 3957.453,E2 3957.453} C_VEL
LIN {X 0,Y 149.534,Z 967.637,A -85,B 0,C 180,E1 3957.312,E2 3957.312} C_VEL
LIN {X 0,Y 142.721,Z 970.993,A -85,B 0,C 180,E1 3956.684,E2 3956.684} C_VEL
LIN {X 0,Y 122.898,Z 980.18,A -85,B 0,C 180,E1 3952.96,E2 3952.96} C_VEL
LIN {X 0,Y 100.376,Z 989.041,A -85,B 0,C 180,E1 3946.757,E2 3946.757} C_VEL
LIN {X 0,Y 81.381,Z 995.353,A -85,B 0,C 180,E1 3938.373,E2 3938.373} C_VEL
LIN {X 0,Y 64.511,Z 1000.054,A -85,B 0,C 180,E1 3925.225,E2 3925.225} C_VEL
LIN {X 0,Y 52.781,Z 1003.154,A -85,B 0,C 180,E1 3905.961,E2 3905.961} C_VEL
LIN {X 0,Y 48.229,Z 1004.542,A -85,B 0,C 180,E1 3883.009,E2 3883.009} C_VEL
LIN {X 0,Y 48.134,Z 1004.822,A -85,B 0,C 180,E1 3870.003,E2 3870.003} C_VEL
LIN {X 0,Y 48.309,Z 1004.504,A -85,B 0,C 180,E1 3855.624,E2 3855.624} C_VEL
LIN {X 0,Y 53.577,Z 1002.884,A -85,B 0,C 180,E1 3831.995,E2 3831.995} C_VEL
LIN {X 0,Y 65.168,Z 999.85,A -85,B 0,C 180,E1 3814.068,E2 3814.068} C_VEL
LIN {X 0,Y 84.116,Z 994.413,A -85,B 0,C 180,E1 3800.132,E2 3800.132} C_VEL
LIN {X 0,Y 103.324,Z 987.943,A -85,B 0,C 180,E1 3792.251,E2 3792.251} C_VEL
LIN {X 0,Y 123.843,Z 979.672,A -85,B 0,C 180,E1 3786.825,E2 3786.825} C_VEL
LIN {X 0,Y 144.169,Z 970.192,A -85,B 0,C 180,E1 3783.082,E2 3783.082} C_VEL
LIN {X 0,Y 164.957,Z 958.701,A -85,B 0,C 180,E1 3780.266,E2 3780.266} C_VEL
LIN {X 0,Y 175.627,Z 952.141,A -85,B 0,C 180,E1 3779.081,E2 3779.081} C_VEL
LIN {X 0,Y 155.239,Z 963.903,A -85,B 0,C 180,E1 3776.549,E2 3776.549} C_VEL
LIN {X 0,Y 135.856,Z 973.442,A -85,B 0,C 180,E1 3773.425,E2 3773.425} C_VEL
LIN {X 0,Y 114.217,Z 982.473,A -85,B 0,C 180,E1 3768.613,E2 3768.613} C_VEL
LIN {X 0,Y 94.534,Z 989.361,A -85,B 0,C 180,E1 3762.132,E2 3762.132} C_VEL
LIN {X 0,Y 75.749,Z 994.714,A -85,B 0,C 180,E1 3752.158,E2 3752.158} C_VEL
LIN {X 0,Y 60.239,Z 998.504,A -85,B 0,C 180,E1 3736.902,E2 3736.902} C_VEL
LIN {X 0,Y 51.029,Z 1000.419,A -85,B 0,C 180,E1 3716.779,E2 3716.779} C_VEL
LIN {X 0,Y 48.378,Z 1001.05,A -85,B 0,C 180,E1 3699.513,E2 3699.513} C_VEL
LIN {X 0,Y 48.157,Z 1001.157,A -85,B 0,C 180,E1 3686.426,E2 3686.426} C_VEL
LIN {X 0,Y 49.752,Z 1000.747,A -85,B 0,C 180,E1 3668.792,E2 3668.792} C_VEL
LIN {X 0,Y 56.996,Z 999.167,A -85,B 0,C 180,E1 3648.195,E2 3648.195} C_VEL
LIN {X 0,Y 71.267,Z 995.951,A -85,B 0,C 180,E1 3631.157,E2 3631.157} C_VEL
LIN {X 0,Y 88.54,Z 991.212,A -85,B 0,C 180,E1 3620.41,E2 3620.41} C_VEL
LIN {X 0,Y 109.612,Z 984.278,A -85,B 0,C 180,E1 3612.592,E2 3612.592} C_VEL
LIN {X 0,Y 129.164,Z 976.533,A -85,B 0,C 180,E1 3607.799,E2 3607.799} C_VEL
LIN {X 0,Y 150.345,Z 966.545,A -85,B 0,C 180,E1 3604.078,E2 3604.078} C_VEL
LIN {X 0,Y 170.016,Z 955.773,A -85,B 0,C 180,E1 3601.479,E2 3601.479} C_VEL
LIN {X 0,Y 175.328,Z 952.486,A -85,B 0,C 180,E1 3600.871,E2 3600.871} C_VEL
LIN {X 0,Y 153.038,Z 965.578,A -85,B 0,C 180,E1 3598.213,E2 3598.213} C_VEL
LIN {X 0,Y 142.721,Z 970.993,A -85,B 0,C 180,E1 3596.684,E2 3596.684} C_VEL
LIN {X 0,Y 135.845,Z 974.248,A -85,B 0,C 180,E1 3595.981,E2 3595.981} C_VEL
LIN {X 0,Y 116.261,Z 982.38,A -85,B 0,C 180,E1 3595.342,E2 3595.342} C_VEL
LIN {X 0,Y 110.27,Z 984.589,A -85,B 0,C 180,E1 3594.448,E2 3594.448} C_VEL
LIN {X 0,Y 88.834,Z 992.025,A -85,B 0,C 180,E1 3588.276,E2 3588.276} C_VEL
LIN {X 0,Y 69.325,Z 997.507,A -85,B 0,C 180,E1 3578.867,E2 3578.867} C_VEL
LIN {X 0,Y 51.297,Z 1001.734,A -85,B 0,C 180,E1 3561.226,E2 3561.226} C_VEL
LIN {X 0,Y 42.225,Z 1003.711,A -85,B 0,C 180,E1 3538.827,E2 3538.827} C_VEL
LIN {X 0,Y 40.083,Z 1004.431,A -85,B 0,C 180,E1 3515.73,E2 3515.73} C_VEL
LIN {X 0,Y 40.087,Z 1004.453,A -85,B 0,C 180,E1 3505.713,E2 3505.713} C_VEL
LIN {X 0,Y 41.849,Z 1003.8,A -85,B 0,C 180,E1 3483.01,E2 3483.01} C_VEL
LIN {X 0,Y 50.102,Z 1001.957,A -85,B 0,C 180,E1 3460.694,E2 3460.694} C_VEL
LIN {X 0,Y 66.614,Z 998.187,A -85,B 0,C 180,E1 3442.968,E2 3442.968} C_VEL
LIN {X 0,Y 85.193,Z 993.034,A -85,B 0,C 180,E1 3433.1,E2 3433.1} C_VEL
LIN {X 0,Y 107.594,Z 985.522,A -85,B 0,C 180,E1 3426.177,E2 3426.177} C_VEL
LIN {X 0,Y 128.049,Z 977.27,A -85,B 0,C 180,E1 3422.09,E2 3422.09} C_VEL
LIN {X 0,Y 149.982,Z 966.729,A -85,B 0,C 180,E1 3418.991,E2 3418.991} C_VEL
LIN {X 0,Y 128.311,Z 976.739,A -85,B 0,C 180,E1 3415.787,E2 3415.787} C_VEL
LIN {X 0,Y 108.125,Z 984.493,A -85,B 0,C 180,E1 3411.616,E2 3411.616} C_VEL
LIN {X 0,Y 86.032,Z 991.454,A -85,B 0,C 180,E1 3404.684,E2 3404.684} C_VEL
LIN {X 0,Y 67.404,Z 996.203,A -85,B 0,C 180,E1 3394.785,E2 3394.785} C_VEL
LIN {X 0,Y 51.212,Z 999.441,A -85,B 0,C 180,E1 3377.882,E2 3377.882} C_VEL
LIN {X 0,Y 42.321,Z 1001.031,A -85,B 0,C 180,E1 3355.16,E2 3355.16} C_VEL
LIN {X 0,Y 40.173,Z 1001.451,A -85,B 0,C 180,E1 3334.278,E2 3334.278} C_VEL
LIN {X 0,Y 40.472,Z 1001.358,A -85,B 0,C 180,E1 3318.598,E2 3318.598} C_VEL
LIN {X 0,Y 44.682,Z 1000.621,A -85,B 0,C 180,E1 3295.984,E2 3295.984} C_VEL
LIN {X 0,Y 57.648,Z 998.279,A -85,B 0,C 180,E1 3273.646,E2 3273.646} C_VEL
LIN {X 0,Y 73.898,Z 994.687,A -85,B 0,C 180,E1 3261.01,E2 3261.01} C_VEL
LIN {X 0,Y 95.05,Z 988.877,A -85,B 0,C 180,E1 3251.982,E2 3251.982} C_VEL
LIN {X 0,Y 114.771,Z 982.194,A -85,B 0,C 180,E1 3246.76,E2 3246.76} C_VEL
LIN {X 0,Y 136.137,Z 973.421,A -85,B 0,C 180,E1 3242.857,E2 3242.857} C_VEL
LIN {X 0,Y 149.69,Z 967.002,A -85,B 0,C 180,E1 3240.96,E2 3240.96} C_VEL
LIN {X 0,Y 127.069,Z 977.78,A -85,B 0,C 180,E1 3237.741,E2 3237.741} C_VEL
LIN {X 0,Y 110.27,Z 984.589,A -85,B 0,C 180,E1 3234.448,E2 3234.448} C_VEL
LIN {X 0,Y 103.216,Z 987.172,A -85,B 0,C 180,E1 3233.326,E2 3233.326} C_VEL
LIN {X 0,Y 83.501,Z 992.91,A -85,B 0,C 180,E1 3231.771,E2 3231.771} C_VEL
LIN {X 0,Y 76.915,Z 994.694,A -85,B 0,C 180,E1 3230.114,E2 3230.114} C_VEL
LIN {X 0,Y 56.684,Z 999.43,A -85,B 0,C 180,E1 3219.197,E2 3219.197} C_VEL
LIN {X 0,Y 40.594,Z 1002.535,A -85,B 0,C 180,E1 3199.777,E2 3199.777} C_VEL
LIN {X 0,Y 32.639,Z 1003.929,A -85,B 0,C 180,E1 3169.695,E2 3169.695} C_VEL
LIN {X 0,Y 32.138,Z 1004.223,A -85,B 0,C 180,E1 3150.005,E2 3150.005} C_VEL
LIN {X 0,Y 32.814,Z 1003.895,A -85,B 0,C 180,E1 3128.561,E2 3128.561} C_VEL
LIN {X 0,Y 41.822,Z 1002.264,A -85,B 0,C 180,E1 3097.928,E2 3097.928} C_VEL
LIN {X 0,Y 57.513,Z 999.224,A -85,B 0,C 180,E1 3080.179,E2 3080.179} C_VEL
LIN {X 0,Y 79.912,Z 993.783,A -85,B 0,C 180,E1 3068.775,E2 3068.775} C_VEL
LIN {X 0,Y 101.537,Z 987.172,A -85,B 0,C 180,E1 3062.821,E2 3062.821} C_VEL
LIN {X 0,Y 123.892,Z 978.663,A -85,B 0,C 180,E1 3058.901,E2 3058.901} C_VEL
LIN {X 0,Y 102.252,Z 986.512,A -85,B 0,C 180,E1 3054.95,E2 3054.95} C_VEL
LIN {X 0,Y 81.427,Z 992.496,A -85,B 0,C 180,E1 3049.171,E2 3049.171} C_VEL
LIN {X 0,Y 60.066,Z 997.342,A -85,B 0,C 180,E1 3038.753,E2 3038.753} C_VEL
LIN {X 0,Y 44.095,Z 1000.064,A -85,B 0,C 180,E1 3022.512,E2 3022.512} C_VEL
LIN {X 0,Y 33.616,Z 1001.564,A -85,B 0,C 180,E1 2992.739,E2 2992.739} C_VEL
LIN {X 0,Y 32.156,Z 1001.811,A -85,B 0,C 180,E1 2969.995,E2 2969.995} C_VEL
LIN {X 0,Y 33.863,Z 1001.553,A -85,B 0,C 180,E1 2945.581,E2 2945.581} C_VEL
LIN {X 0,Y 44.735,Z 999.99,A -85,B 0,C 180,E1 2916.429,E2 2916.429} C_VEL
LIN {X 0,Y 61.733,Z 997.085,A -85,B 0,C 180,E1 2900.06,E2 2900.06} C_VEL
LIN {X 0,Y 82.343,Z 992.318,A -85,B 0,C 180,E1 2890.43,E2 2890.43} C_VEL
LIN {X 0,Y 103.329,Z 986.258,A -85,B 0,C 180,E1 2884.735,E2 2884.735} C_VEL
LIN {X 0,Y 123.642,Z 978.864,A -85,B 0,C 180,E1 2881.058,E2 2881.058} C_VEL
LIN {X 0,Y 101.565,Z 987.236,A -85,B 0,C 180,E1 2877.18,E2 2877.18} C_VEL
LIN {X 0,Y 80.506,Z 993.674,A -85,B 0,C 180,E1 2871.431,E2 2871.431} C_VEL
LIN {X 0,Y 76.915,Z 994.694,A -85,B 0,C 180,E1 2870.114,E2 2870.114} C_VEL
LIN {X 0,Y 69.842,Z 996.486,A -85,B 0,C 180,E1 2868.035,E2 2868.035} C_VEL
LIN {X 0,Y 49.453,Z 1000.155,A -85,B 0,C 180,E1 2863.3,E2 2863.3} C_VEL
LIN {X 0,Y 43.6,Z 1001.008,A -85,B 0,C 180,E1 2859.473,E2 2859.473} C_VEL
LIN {X 0,Y 29.309,Z 1003.047,A -85,B 0,C 180,E1 2835.759,E2 2835.759} C_VEL
LIN {X 0,Y 24.109,Z 1003.827,A -85,B 0,C 180,E1 2799.555,E2 2799.555} C_VEL
LIN {X 0,Y 24.091,Z 1003.872,A -85,B 0,C 180,E1 2784.856,E2 2784.856} C_VEL
LIN {X 0,Y 28.244,Z 1003.185,A -85,B 0,C 180,E1 2747.745,E2 2747.745} C_VEL
LIN {X 0,Y 42.068,Z 1001.21,A -85,B 0,C 180,E1 2722.064,E2 2722.064} C_VEL
LIN {X 0,Y 63.592,Z 997.2,A -85,B 0,C 180,E1 2707.947,E2 2707.947} C_VEL
LIN {X 0,Y 84.724,Z 991.944,A -85,B 0,C 180,E1 2701.351,E2 2701.351} C_VEL
LIN {X 0,Y 97.241,Z 988.178,A -85,B 0,C 180,E1 2698.778,E2 2698.778} C_VEL
LIN {X 0,Y 75.45,Z 994.025,A -85,B 0,C 180,E1 2693.587,E2 2693.587} C_VEL
LIN {X 0,Y 53.983,Z 998.251,A -85,B 0,C 180,E1 2684.36,E2 2684.36} C_VEL
LIN {X 0,Y 35.908,Z 1000.896,A -85,B 0,C 180,E1 2666.634,E2 2666.634} C_VEL
LIN {X 0,Y 25.412,Z 1001.918,A -85,B 0,C 180,E1 2633.161,E2 2633.161} C_VEL
LIN {X 0,Y 24.158,Z 1002.099,A -85,B 0,C 180,E1 2607.622,E2 2607.622} C_VEL
LIN {X 0,Y 27.539,Z 1001.781,A -85,B 0,C 180,E1 2574.483,E2 2574.483} C_VEL
LIN {X 0,Y 41.202,Z 1000.192,A -85,B 0,C 180,E1 2546.123,E2 2546.123} C_VEL
LIN {X 0,Y 61.258,Z 997.073,A -85,B 0,C 180,E1 2531.69,E2 2531.69} C_VEL
LIN {X 0,Y 83.203,Z 992.14,A -85,B 0,C 180,E1 2524.179,E2 2524.179} C_VEL
LIN {X 0,Y 96.998,Z 988.329,A -85,B 0,C 180,E1 2521.156,E2 2521.156} C_VEL
LIN {X 0,Y 74.18,Z 994.845,A -85,B 0,C 180,E1 2515.835,E2 2515.835} C_VEL
LIN {X 0,Y 52.471,Z 999.459,A -85,B 0,C 180,E1 2506.351,E2 2506.351} C_VEL
LIN {X 0,Y 43.6,Z 1001.008,A -85,B 0,C 180,E1 2499.473,E2 2499.473} C_VEL
LIN {X 0,Y 37.006,Z 1001.929,A -85,B 0,C 180,E1 2493.761,E2 2493.761} C_VEL
LIN {X 0,Y 24.225,Z 1003.028,A -85,B 0,C 180,E1 2480.505,E2 2480.505} C_VEL
LIN {X 0,Y 17.155,Z 1003.424,A -85,B 0,C 180,E1 2457.934,E2 2457.934} C_VEL
LIN {X 0,Y 16.367,Z 1003.489,A -85,B 0,C 180,E1 2448.734,E2 2448.734} C_VEL
LIN {X 0,Y 16.099,Z 1003.601,A -85,B 0,C 180,E1 2426.45,E2 2426.45} C_VEL
LIN {X 0,Y 21.963,Z 1002.976,A -85,B 0,C 180,E1 2376.279,E2 2376.279} C_VEL
LIN {X 0,Y 38.775,Z 1001.022,A -85,B 0,C 180,E1 2351.566,E2 2351.566} C_VEL
LIN {X 0,Y 61.133,Z 997.29,A -85,B 0,C 180,E1 2340.935,E2 2340.935} C_VEL
LIN {X 0,Y 69.613,Z 995.443,A -85,B 0,C 180,E1 2338.664,E2 2338.664} C_VEL
LIN {X 0,Y 48.543,Z 999.161,A -85,B 0,C 180,E1 2331.301,E2 2331.301} C_VEL
LIN {X 0,Y 27.998,Z 1001.519,A -85,B 0,C 180,E1 2313.2,E2 2313.2} C_VEL
LIN {X 0,Y 17.485,Z 1002.257,A -85,B 0,C 180,E1 2277.21,E2 2277.21} C_VEL
LIN {X 0,Y 16.217,Z 1002.378,A -85,B 0,C 180,E1 2242.908,E2 2242.908} C_VEL
LIN {X 0,Y 22.106,Z 1002.023,A -85,B 0,C 180,E1 2199.74,E2 2199.74} C_VEL
LIN {X 0,Y 38.306,Z 1000.499,A -85,B 0,C 180,E1 2175.042,E2 2175.042} C_VEL
LIN {X 0,Y 60.131,Z 997.382,A -85,B 0,C 180,E1 2163.966,E2 2163.966} C_VEL
LIN {X 0,Y 69.454,Z 995.527,A -85,B 0,C 180,E1 2161.295,E2 2161.295} C_VEL
LIN {X 0,Y 47.279,Z 999.83,A -85,B 0,C 180,E1 2153.665,E2 2153.665} C_VEL
LIN {X 0,Y 26.606,Z 1002.507,A -85,B 0,C 180,E1 2134.413,E2 2134.413} C_VEL
LIN {X 0,Y 16.735,Z 1003.438,A -85,B 0,C 180,E1 2094.729,E2 2094.729} C_VEL
LIN {X 0,Y 16.367,Z 1003.489,A -85,B 0,C 180,E1 2088.734,E2 2088.734} C_VEL
LIN {X 0,Y 15.398,Z 1003.593,A -85,B 0,C 180,E1 2069.317,E2 2069.317} C_VEL
LIN {X 0,Y 14.86,Z 1003.391,A -85,B 0,C 180,E1 2041.874,E2 2041.874} C_VEL
LIN {X 0,Y 23.904,Z 1002.235,A -85,B 0,C 180,E1 1989.05,E2 1989.05} C_VEL
LIN {X 0,Y 28.062,Z 1001.872,A -85,B 0,C 180,E1 1984.53,E2 1984.53} C_VEL
LIN {X 0,Y 39.84,Z 1000.48,A -85,B 0,C 180,E1 1978.379,E2 1978.379} C_VEL
LIN {X 0,Y 20.728,Z 1002.127,A -85,B 0,C 180,E1 1964.682,E2 1964.682} C_VEL
LIN {X 0,Y 8.563,Z 1002.652,A -85,B 0,C 180,E1 1910.483,E2 1910.483} C_VEL
LIN {X 0,Y 9.294,Z 1002.62,A -85,B 0,C 180,E1 1857.442,E2 1857.442} C_VEL
LIN {X 0,Y 22.569,Z 1002.024,A -85,B 0,C 180,E1 1812.922,E2 1812.922} C_VEL
LIN {X 0,Y 39.673,Z 1000.531,A -85,B 0,C 180,E1 1801.447,E2 1801.447} C_VEL
LIN {X 0,Y 20.443,Z 1002.508,A -85,B 0,C 180,E1 1788.013,E2 1788.013} C_VEL
LIN {X 0,Y 8.158,Z 1003.278,A -85,B 0,C 180,E1 1724.208,E2 1724.208} C_VEL
LIN {X 0,Y 8.161,Z 1003.273,A -85,B 0,C 180,E1 1695.837,E2 1695.837} C_VEL
LIN {X 0,Y 20.438,Z 1002.492,A -85,B 0,C 180,E1 1631.99,E2 1631.99} C_VEL
LIN {X 0,Y 28.062,Z 1001.872,A -85,B 0,C 180,E1 1624.53,E2 1624.53} C_VEL
LIN {X 0,Y 27.023,Z 1001.91,A -85,B 0,C 180,E1 1622.442,E2 1622.442} C_VEL
LIN {X 0,Y 20.993,Z 1002.26,A -85,B 0,C 180,E1 1619.657,E2 1619.657} C_VEL
LIN {X 0,Y 5.63,Z 1002.903,A -85,B 0,C 180,E1 1616.232,E2 1616.232} C_VEL
LIN {X 0,Y 0.511,Z 1003.009,A -85,B 0,C 180,E1 1624.234,E2 1624.234} C_VEL
LIN {X 0,Y 1.379,Z 1002.993,A -85,B 0,C 180,E1 1803.262,E2 1803.262} C_VEL
LIN {X 0,Y 1.388,Z 1002.987,A -85,B 0,C 180,E1 1976.776,E2 1976.776} C_VEL
LIN {X 0,Y 0.511,Z 1003.009,A -85,B 0,C 180,E1 1984.234,E2 1984.234} C_VEL
LIN {X 0,Y 1.457,Z 1005.009,A -85,B 0,C 180,E1 2149.71,E2 2149.71} C_VEL
LIN {X 0,Y 1.457,Z 1028,A -85,B 0,C 180,E1 2149.71,E2 2149.71} C_VEL
LIN {X 0,Y 1.457,Z 1028,A -85,B 0,C 180,E1 2149.71,E2 2149.71}

QRS_NEXT_CUT()

QRS_NEXT()
QRS_HOME()

END
